// TIA Portal V17 export
// export: Created 2023-09-06T09:59:09.1457623Z, ExportSetting WithDefaults, DisplayName Totally Integrated Automation Portal, DisplayVersion V17 Update 6, DisplayName TIA Portal Openness, DisplayVersion V17 Update 6, DisplayName TIA Portal Teamcenter Gateway, DisplayVersion V17 Update 6, DisplayName TIA Portal Version Control Interface, DisplayVersion V17, DisplayName Simotion SCOUT TIA, DisplayVersion 5.4.3.0, DisplayName TIA Portal Test Suite Advanced, DisplayVersion V17 Update 1, DisplayName SIMOCODE ES, DisplayVersion V17 Update 5, DisplayName SINAMICS Startdrive Advanced, DisplayVersion V17 SP1, DisplayName SINAMICS Startdrive G130, G150, S120, S150, SINAMICS MV, S210, DisplayVersion V17 SP1, DisplayName SINAMICS Startdrive G110M, G120, G120C, G120D, G120P, G115D, DisplayVersion V17 SP1, DisplayName SIRIUS Safety ES, DisplayVersion V17 Update 5, DisplayName STEP 7 Professional, DisplayVersion V17 Update 6, DisplayName STEP 7 CFC, DisplayVersion V17 Update 1, DisplayName STEP 7 Safety, DisplayVersion V17 Update 6, DisplayName WinCC Advanced, DisplayVersion V17 Update 6, DisplayName SIMATIC Visualization Architect, DisplayVersion V17 Update 5
FUNCTION "05_Output Feedback" : Void   // FC6, F_FBD
TITLE = Manage Safety Outputs
{ S7_Optimized_Access := 'TRUE' }
VERSION : 0.1
// stored: AutoNumber true, IsIECCheckEnabled false, UDAEnableTagReadback false
   VAR_TEMP
      DU_EX : Bool;
      ISPC_EX : Bool;
      ZONE_EX : Bool;
   END_VAR
BEGIN

REGION Network 1: Area S1 =SC01+DU001/DU019.EL001 DRIVE UNIT DU001/DU019
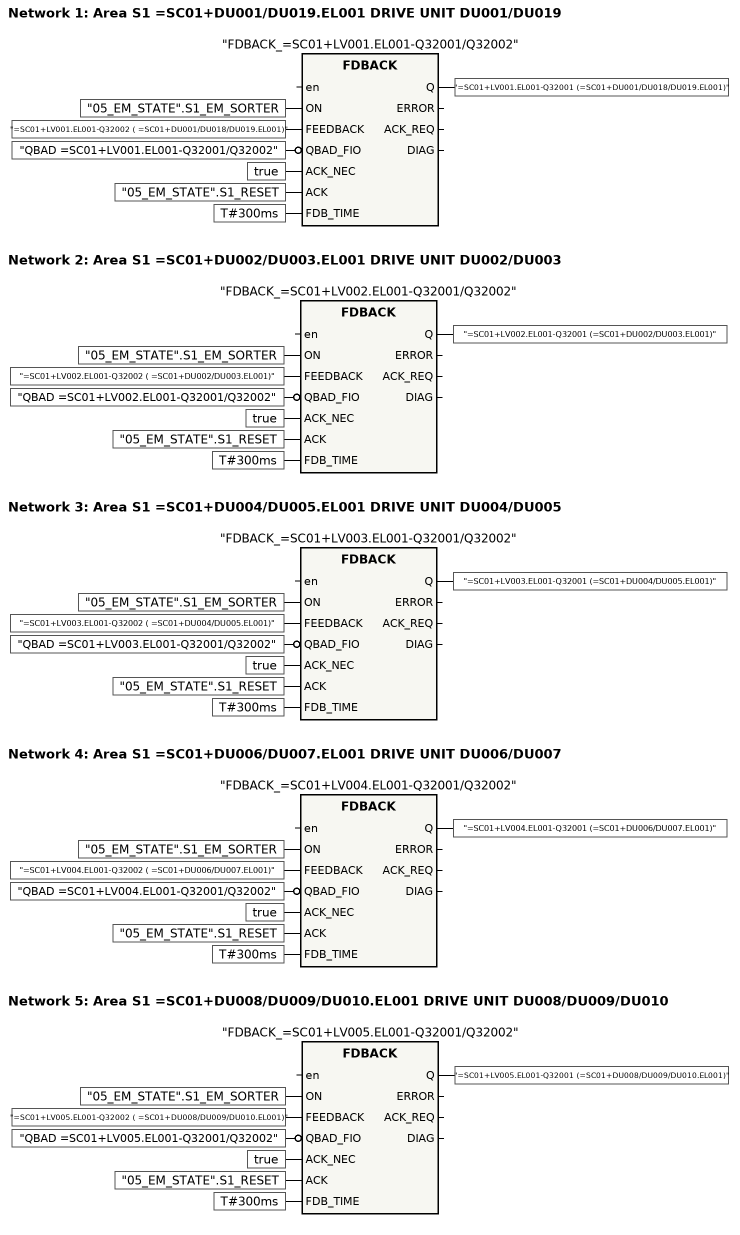
   "FDBACK_=SC01+LV001.EL001-Q32001/Q32002"(ON := "05_EM_STATE".S1_EM_SORTER,   // FDBACK
                           FEEDBACK := "=SC01+LV001.EL001-Q32002 ( =SC01+DU001/DU018/DU019.EL001)",
                           QBAD_FIO := NOT "QBAD =SC01+LV001.EL001-Q32001/Q32002",
                           ACK_NEC := true,
                           ACK := "05_EM_STATE".S1_RESET,
                           FDB_TIME := T#300ms,
                           Q => "=SC01+LV001.EL001-Q32001 (=SC01+DU001/DU018/DU019.EL001)");
END_REGION

REGION Network 2: Area S1 =SC01+DU002/DU003.EL001 DRIVE UNIT DU002/DU003
   "FDBACK_=SC01+LV002.EL001-Q32001/Q32002"(ON := "05_EM_STATE".S1_EM_SORTER,   // FDBACK
                           FEEDBACK := "=SC01+LV002.EL001-Q32002 ( =SC01+DU002/DU003.EL001)",
                           QBAD_FIO := NOT "QBAD =SC01+LV002.EL001-Q32001/Q32002",
                           ACK_NEC := true,
                           ACK := "05_EM_STATE".S1_RESET,
                           FDB_TIME := T#300ms,
                           Q => "=SC01+LV002.EL001-Q32001 (=SC01+DU002/DU003.EL001)");
END_REGION

REGION Network 3: Area S1 =SC01+DU004/DU005.EL001 DRIVE UNIT DU004/DU005
   "FDBACK_=SC01+LV003.EL001-Q32001/Q32002"(ON := "05_EM_STATE".S1_EM_SORTER,   // FDBACK
                           FEEDBACK := "=SC01+LV003.EL001-Q32002 ( =SC01+DU004/DU005.EL001)",
                           QBAD_FIO := NOT "QBAD =SC01+LV003.EL001-Q32001/Q32002",
                           ACK_NEC := true,
                           ACK := "05_EM_STATE".S1_RESET,
                           FDB_TIME := T#300ms,
                           Q => "=SC01+LV003.EL001-Q32001 (=SC01+DU004/DU005.EL001)");
END_REGION

REGION Network 4: Area S1 =SC01+DU006/DU007.EL001 DRIVE UNIT DU006/DU007
   "FDBACK_=SC01+LV004.EL001-Q32001/Q32002"(ON := "05_EM_STATE".S1_EM_SORTER,   // FDBACK
                           FEEDBACK := "=SC01+LV004.EL001-Q32002 ( =SC01+DU006/DU007.EL001)",
                           QBAD_FIO := NOT "QBAD =SC01+LV004.EL001-Q32001/Q32002",
                           ACK_NEC := true,
                           ACK := "05_EM_STATE".S1_RESET,
                           FDB_TIME := T#300ms,
                           Q => "=SC01+LV004.EL001-Q32001 (=SC01+DU006/DU007.EL001)");
END_REGION

REGION Network 5: Area S1 =SC01+DU008/DU009/DU010.EL001 DRIVE UNIT DU008/DU009/DU010
   "FDBACK_=SC01+LV005.EL001-Q32001/Q32002"(ON := "05_EM_STATE".S1_EM_SORTER,   // FDBACK
                           FEEDBACK := "=SC01+LV005.EL001-Q32002 ( =SC01+DU008/DU009/DU010.EL001)",
                           QBAD_FIO := NOT "QBAD =SC01+LV005.EL001-Q32001/Q32002",
                           ACK_NEC := true,
                           ACK := "05_EM_STATE".S1_RESET,
                           FDB_TIME := T#300ms,
                           Q => "=SC01+LV005.EL001-Q32001 (=SC01+DU008/DU009/DU010.EL001)");
END_REGION

REGION Network 6: Area S1 =SC01+DU011/DU012/DU013.EL001 DRIVE UNIT DU011/DU012/DU013
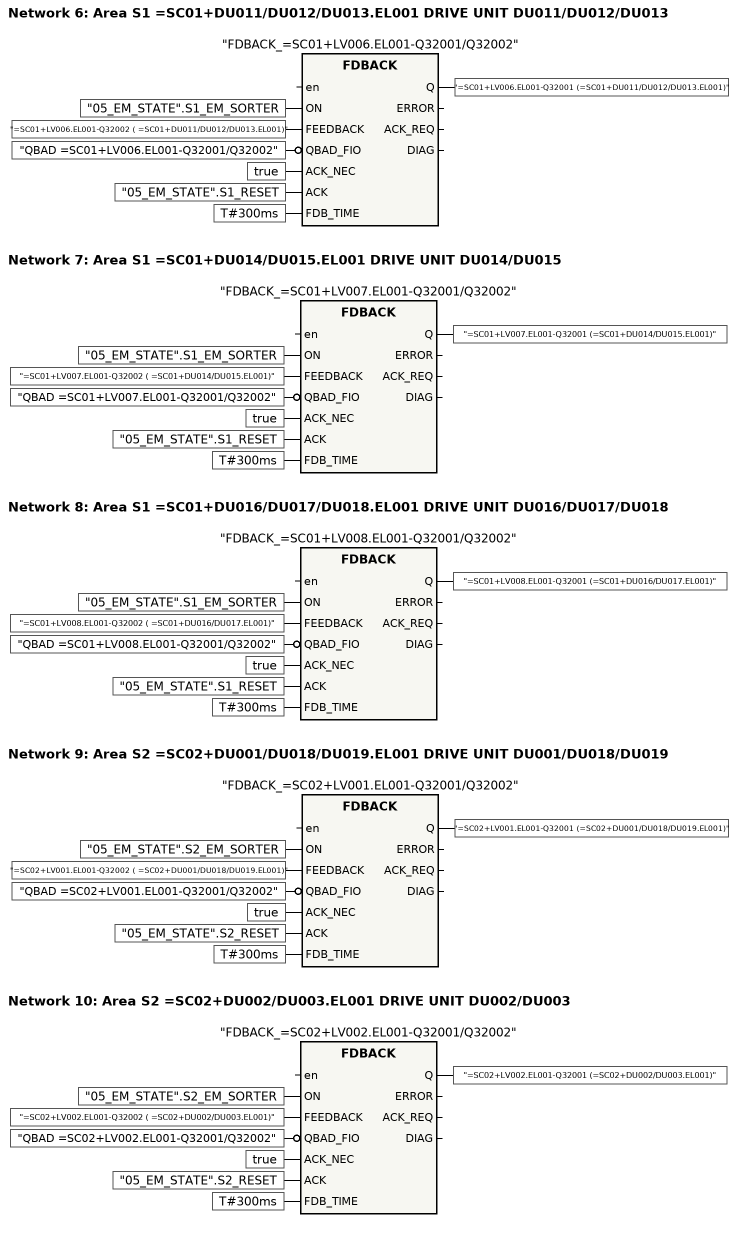
   "FDBACK_=SC01+LV006.EL001-Q32001/Q32002"(ON := "05_EM_STATE".S1_EM_SORTER,   // FDBACK
                           FEEDBACK := "=SC01+LV006.EL001-Q32002 ( =SC01+DU011/DU012/DU013.EL001)",
                           QBAD_FIO := NOT "QBAD =SC01+LV006.EL001-Q32001/Q32002",
                           ACK_NEC := true,
                           ACK := "05_EM_STATE".S1_RESET,
                           FDB_TIME := T#300ms,
                           Q => "=SC01+LV006.EL001-Q32001 (=SC01+DU011/DU012/DU013.EL001)");
END_REGION

REGION Network 7: Area S1 =SC01+DU014/DU015.EL001 DRIVE UNIT DU014/DU015
   "FDBACK_=SC01+LV007.EL001-Q32001/Q32002"(ON := "05_EM_STATE".S1_EM_SORTER,   // FDBACK
                           FEEDBACK := "=SC01+LV007.EL001-Q32002 ( =SC01+DU014/DU015.EL001)",
                           QBAD_FIO := NOT "QBAD =SC01+LV007.EL001-Q32001/Q32002",
                           ACK_NEC := true,
                           ACK := "05_EM_STATE".S1_RESET,
                           FDB_TIME := T#300ms,
                           Q => "=SC01+LV007.EL001-Q32001 (=SC01+DU014/DU015.EL001)");
END_REGION

REGION Network 8: Area S1 =SC01+DU016/DU017/DU018.EL001 DRIVE UNIT DU016/DU017/DU018
   "FDBACK_=SC01+LV008.EL001-Q32001/Q32002"(ON := "05_EM_STATE".S1_EM_SORTER,   // FDBACK
                           FEEDBACK := "=SC01+LV008.EL001-Q32002 ( =SC01+DU016/DU017.EL001)",
                           QBAD_FIO := NOT "QBAD =SC01+LV008.EL001-Q32001/Q32002",
                           ACK_NEC := true,
                           ACK := "05_EM_STATE".S1_RESET,
                           FDB_TIME := T#300ms,
                           Q => "=SC01+LV008.EL001-Q32001 (=SC01+DU016/DU017.EL001)");
END_REGION

REGION Network 9: Area S2 =SC02+DU001/DU018/DU019.EL001 DRIVE UNIT DU001/DU018/DU019
   "FDBACK_=SC02+LV001.EL001-Q32001/Q32002"(ON := "05_EM_STATE".S2_EM_SORTER,   // FDBACK
                           FEEDBACK := "=SC02+LV001.EL001-Q32002 ( =SC02+DU001/DU018/DU019.EL001)",
                           QBAD_FIO := NOT "QBAD =SC02+LV001.EL001-Q32001/Q32002",
                           ACK_NEC := true,
                           ACK := "05_EM_STATE".S2_RESET,
                           FDB_TIME := T#300ms,
                           Q => "=SC02+LV001.EL001-Q32001 (=SC02+DU001/DU018/DU019.EL001)");
END_REGION

REGION Network 10: Area S2 =SC02+DU002/DU003.EL001 DRIVE UNIT DU002/DU003
   "FDBACK_=SC02+LV002.EL001-Q32001/Q32002"(ON := "05_EM_STATE".S2_EM_SORTER,   // FDBACK
                           FEEDBACK := "=SC02+LV002.EL001-Q32002 ( =SC02+DU002/DU003.EL001)",
                           QBAD_FIO := NOT "QBAD =SC02+LV002.EL001-Q32001/Q32002",
                           ACK_NEC := true,
                           ACK := "05_EM_STATE".S2_RESET,
                           FDB_TIME := T#300ms,
                           Q => "=SC02+LV002.EL001-Q32001 (=SC02+DU002/DU003.EL001)");
END_REGION

REGION Network 11: Area S2 =SC02+DU004/DU005.EL001 DRIVE UNIT DU004/DU005
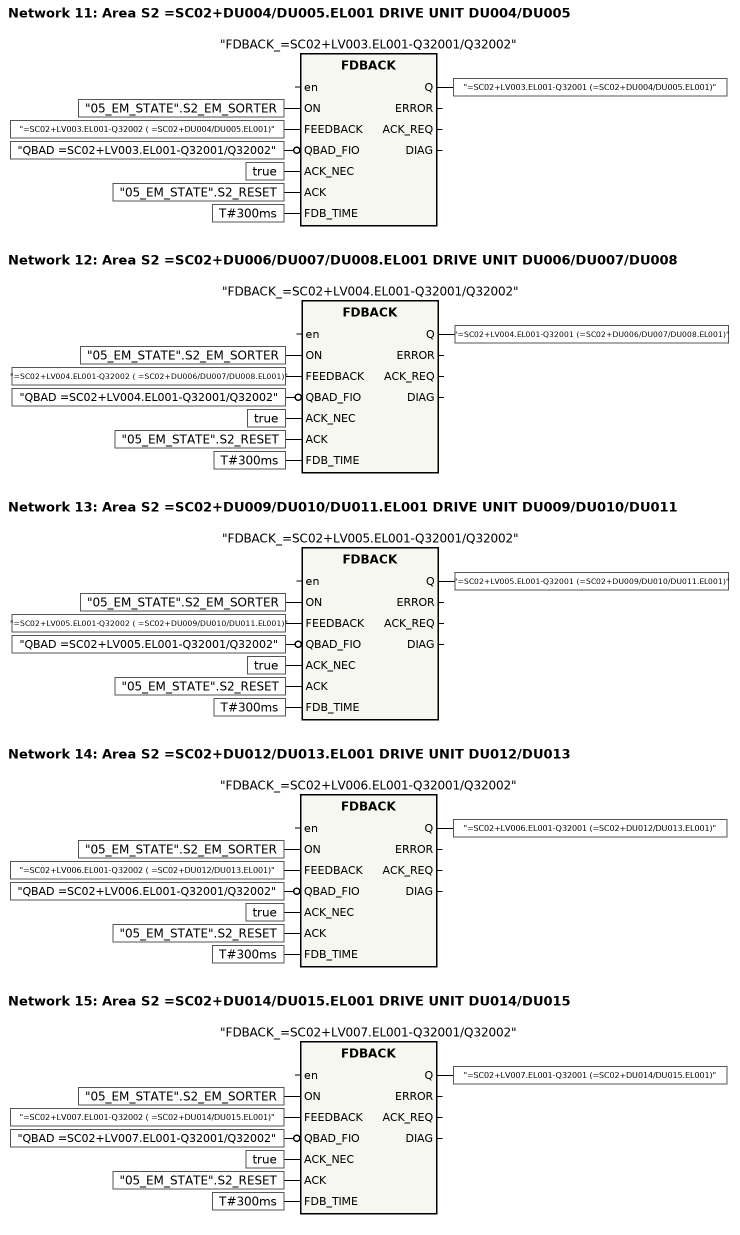
   "FDBACK_=SC02+LV003.EL001-Q32001/Q32002"(ON := "05_EM_STATE".S2_EM_SORTER,   // FDBACK
                           FEEDBACK := "=SC02+LV003.EL001-Q32002 ( =SC02+DU004/DU005.EL001)",
                           QBAD_FIO := NOT "QBAD =SC02+LV003.EL001-Q32001/Q32002",
                           ACK_NEC := true,
                           ACK := "05_EM_STATE".S2_RESET,
                           FDB_TIME := T#300ms,
                           Q => "=SC02+LV003.EL001-Q32001 (=SC02+DU004/DU005.EL001)");
END_REGION

REGION Network 12: Area S2 =SC02+DU006/DU007/DU008.EL001 DRIVE UNIT DU006/DU007/DU008
   "FDBACK_=SC02+LV004.EL001-Q32001/Q32002"(ON := "05_EM_STATE".S2_EM_SORTER,   // FDBACK
                           FEEDBACK := "=SC02+LV004.EL001-Q32002 ( =SC02+DU006/DU007/DU008.EL001)",
                           QBAD_FIO := NOT "QBAD =SC02+LV004.EL001-Q32001/Q32002",
                           ACK_NEC := true,
                           ACK := "05_EM_STATE".S2_RESET,
                           FDB_TIME := T#300ms,
                           Q => "=SC02+LV004.EL001-Q32001 (=SC02+DU006/DU007/DU008.EL001)");
END_REGION

REGION Network 13: Area S2 =SC02+DU009/DU010/DU011.EL001 DRIVE UNIT DU009/DU010/DU011
   "FDBACK_=SC02+LV005.EL001-Q32001/Q32002"(ON := "05_EM_STATE".S2_EM_SORTER,   // FDBACK
                           FEEDBACK := "=SC02+LV005.EL001-Q32002 ( =SC02+DU009/DU010/DU011.EL001)",
                           QBAD_FIO := NOT "QBAD =SC02+LV005.EL001-Q32001/Q32002",
                           ACK_NEC := true,
                           ACK := "05_EM_STATE".S2_RESET,
                           FDB_TIME := T#300ms,
                           Q => "=SC02+LV005.EL001-Q32001 (=SC02+DU009/DU010/DU011.EL001)");
END_REGION

REGION Network 14: Area S2 =SC02+DU012/DU013.EL001 DRIVE UNIT DU012/DU013
   "FDBACK_=SC02+LV006.EL001-Q32001/Q32002"(ON := "05_EM_STATE".S2_EM_SORTER,   // FDBACK
                           FEEDBACK := "=SC02+LV006.EL001-Q32002 ( =SC02+DU012/DU013.EL001)",
                           QBAD_FIO := NOT "QBAD =SC02+LV006.EL001-Q32001/Q32002",
                           ACK_NEC := true,
                           ACK := "05_EM_STATE".S2_RESET,
                           FDB_TIME := T#300ms,
                           Q => "=SC02+LV006.EL001-Q32001 (=SC02+DU012/DU013.EL001)");
END_REGION

REGION Network 15: Area S2 =SC02+DU014/DU015.EL001 DRIVE UNIT DU014/DU015
   "FDBACK_=SC02+LV007.EL001-Q32001/Q32002"(ON := "05_EM_STATE".S2_EM_SORTER,   // FDBACK
                           FEEDBACK := "=SC02+LV007.EL001-Q32002 ( =SC02+DU014/DU015.EL001)",
                           QBAD_FIO := NOT "QBAD =SC02+LV007.EL001-Q32001/Q32002",
                           ACK_NEC := true,
                           ACK := "05_EM_STATE".S2_RESET,
                           FDB_TIME := T#300ms,
                           Q => "=SC02+LV007.EL001-Q32001 (=SC02+DU014/DU015.EL001)");
END_REGION

REGION Network 16: Area S2 =SC02+DU016/DU017.EL001 DRIVE UNIT DU016/DU017
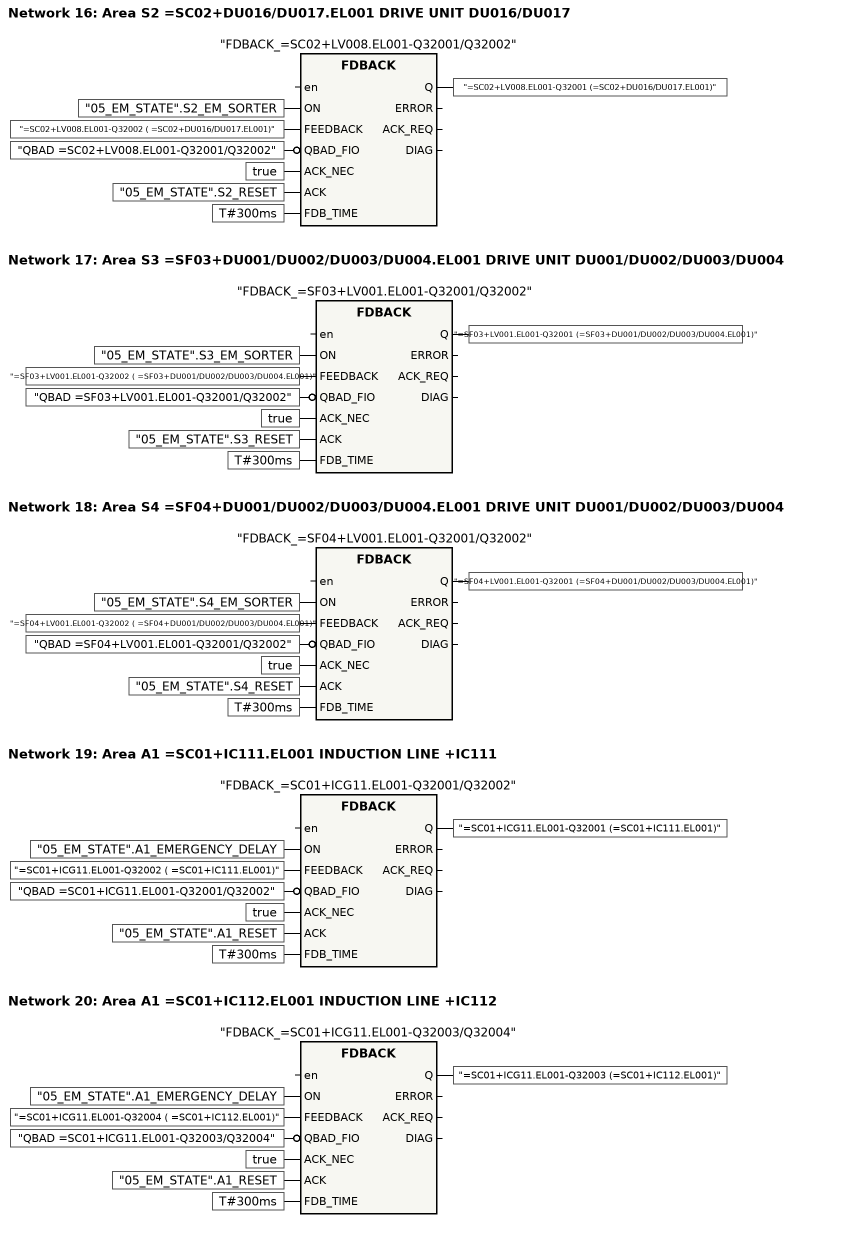
   "FDBACK_=SC02+LV008.EL001-Q32001/Q32002"(ON := "05_EM_STATE".S2_EM_SORTER,   // FDBACK
                           FEEDBACK := "=SC02+LV008.EL001-Q32002 ( =SC02+DU016/DU017.EL001)",
                           QBAD_FIO := NOT "QBAD =SC02+LV008.EL001-Q32001/Q32002",
                           ACK_NEC := true,
                           ACK := "05_EM_STATE".S2_RESET,
                           FDB_TIME := T#300ms,
                           Q => "=SC02+LV008.EL001-Q32001 (=SC02+DU016/DU017.EL001)");
END_REGION

REGION Network 17: Area S3 =SF03+DU001/DU002/DU003/DU004.EL001 DRIVE UNIT DU001/DU002/DU003/DU004
   "FDBACK_=SF03+LV001.EL001-Q32001/Q32002"(ON := "05_EM_STATE".S3_EM_SORTER,   // FDBACK
                           FEEDBACK := "=SF03+LV001.EL001-Q32002 ( =SF03+DU001/DU002/DU003/DU004.EL001)",
                           QBAD_FIO := NOT "QBAD =SF03+LV001.EL001-Q32001/Q32002",
                           ACK_NEC := true,
                           ACK := "05_EM_STATE".S3_RESET,
                           FDB_TIME := T#300ms,
                           Q => "=SF03+LV001.EL001-Q32001 (=SF03+DU001/DU002/DU003/DU004.EL001)");
END_REGION

REGION Network 18: Area S4 =SF04+DU001/DU002/DU003/DU004.EL001 DRIVE UNIT DU001/DU002/DU003/DU004
   "FDBACK_=SF04+LV001.EL001-Q32001/Q32002"(ON := "05_EM_STATE".S4_EM_SORTER,   // FDBACK
                           FEEDBACK := "=SF04+LV001.EL001-Q32002 ( =SF04+DU001/DU002/DU003/DU004.EL001)",
                           QBAD_FIO := NOT "QBAD =SF04+LV001.EL001-Q32001/Q32002",
                           ACK_NEC := true,
                           ACK := "05_EM_STATE".S4_RESET,
                           FDB_TIME := T#300ms,
                           Q => "=SF04+LV001.EL001-Q32001 (=SF04+DU001/DU002/DU003/DU004.EL001)");
END_REGION

REGION Network 19: Area A1 =SC01+IC111.EL001 INDUCTION LINE +IC111
   "FDBACK_=SC01+ICG11.EL001-Q32001/Q32002"(ON := "05_EM_STATE".A1_EMERGENCY_DELAY,   // FDBACK
                           FEEDBACK := "=SC01+ICG11.EL001-Q32002 ( =SC01+IC111.EL001)",
                           QBAD_FIO := NOT "QBAD =SC01+ICG11.EL001-Q32001/Q32002",
                           ACK_NEC := true,
                           ACK := "05_EM_STATE".A1_RESET,
                           FDB_TIME := T#300ms,
                           Q => "=SC01+ICG11.EL001-Q32001 (=SC01+IC111.EL001)");
END_REGION

REGION Network 20: Area A1 =SC01+IC112.EL001 INDUCTION LINE +IC112
   "FDBACK_=SC01+ICG11.EL001-Q32003/Q32004"(ON := "05_EM_STATE".A1_EMERGENCY_DELAY,   // FDBACK
                           FEEDBACK := "=SC01+ICG11.EL001-Q32004 ( =SC01+IC112.EL001)",
                           QBAD_FIO := NOT "QBAD =SC01+ICG11.EL001-Q32003/Q32004",
                           ACK_NEC := true,
                           ACK := "05_EM_STATE".A1_RESET,
                           FDB_TIME := T#300ms,
                           Q => "=SC01+ICG11.EL001-Q32003 (=SC01+IC112.EL001)");
END_REGION

REGION Network 21: Area A1 =SC01+IC113.EL001 INDUCTION LINE +IC113
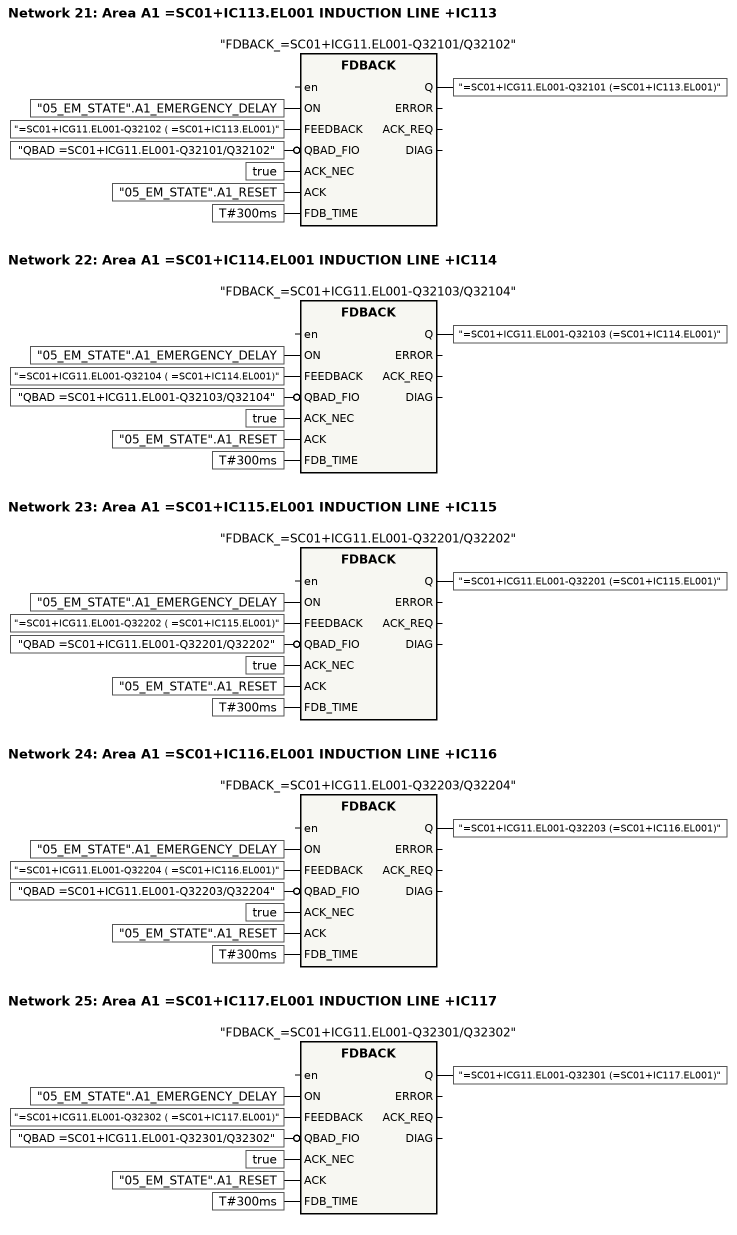
   "FDBACK_=SC01+ICG11.EL001-Q32101/Q32102"(ON := "05_EM_STATE".A1_EMERGENCY_DELAY,   // FDBACK
                           FEEDBACK := "=SC01+ICG11.EL001-Q32102 ( =SC01+IC113.EL001)",
                           QBAD_FIO := NOT "QBAD =SC01+ICG11.EL001-Q32101/Q32102",
                           ACK_NEC := true,
                           ACK := "05_EM_STATE".A1_RESET,
                           FDB_TIME := T#300ms,
                           Q => "=SC01+ICG11.EL001-Q32101 (=SC01+IC113.EL001)");
END_REGION

REGION Network 22: Area A1 =SC01+IC114.EL001 INDUCTION LINE +IC114
   "FDBACK_=SC01+ICG11.EL001-Q32103/Q32104"(ON := "05_EM_STATE".A1_EMERGENCY_DELAY,   // FDBACK
                           FEEDBACK := "=SC01+ICG11.EL001-Q32104 ( =SC01+IC114.EL001)",
                           QBAD_FIO := NOT "QBAD =SC01+ICG11.EL001-Q32103/Q32104",
                           ACK_NEC := true,
                           ACK := "05_EM_STATE".A1_RESET,
                           FDB_TIME := T#300ms,
                           Q => "=SC01+ICG11.EL001-Q32103 (=SC01+IC114.EL001)");
END_REGION

REGION Network 23: Area A1 =SC01+IC115.EL001 INDUCTION LINE +IC115
   "FDBACK_=SC01+ICG11.EL001-Q32201/Q32202"(ON := "05_EM_STATE".A1_EMERGENCY_DELAY,   // FDBACK
                           FEEDBACK := "=SC01+ICG11.EL001-Q32202 ( =SC01+IC115.EL001)",
                           QBAD_FIO := NOT "QBAD =SC01+ICG11.EL001-Q32201/Q32202",
                           ACK_NEC := true,
                           ACK := "05_EM_STATE".A1_RESET,
                           FDB_TIME := T#300ms,
                           Q => "=SC01+ICG11.EL001-Q32201 (=SC01+IC115.EL001)");
END_REGION

REGION Network 24: Area A1 =SC01+IC116.EL001 INDUCTION LINE +IC116
   "FDBACK_=SC01+ICG11.EL001-Q32203/Q32204"(ON := "05_EM_STATE".A1_EMERGENCY_DELAY,   // FDBACK
                           FEEDBACK := "=SC01+ICG11.EL001-Q32204 ( =SC01+IC116.EL001)",
                           QBAD_FIO := NOT "QBAD =SC01+ICG11.EL001-Q32203/Q32204",
                           ACK_NEC := true,
                           ACK := "05_EM_STATE".A1_RESET,
                           FDB_TIME := T#300ms,
                           Q => "=SC01+ICG11.EL001-Q32203 (=SC01+IC116.EL001)");
END_REGION

REGION Network 25: Area A1 =SC01+IC117.EL001 INDUCTION LINE +IC117
   "FDBACK_=SC01+ICG11.EL001-Q32301/Q32302"(ON := "05_EM_STATE".A1_EMERGENCY_DELAY,   // FDBACK
                           FEEDBACK := "=SC01+ICG11.EL001-Q32302 ( =SC01+IC117.EL001)",
                           QBAD_FIO := NOT "QBAD =SC01+ICG11.EL001-Q32301/Q32302",
                           ACK_NEC := true,
                           ACK := "05_EM_STATE".A1_RESET,
                           FDB_TIME := T#300ms,
                           Q => "=SC01+ICG11.EL001-Q32301 (=SC01+IC117.EL001)");
END_REGION

REGION Network 26: Area A1 =SC01+IC121.EL001 INDUCTION LINE +IC121
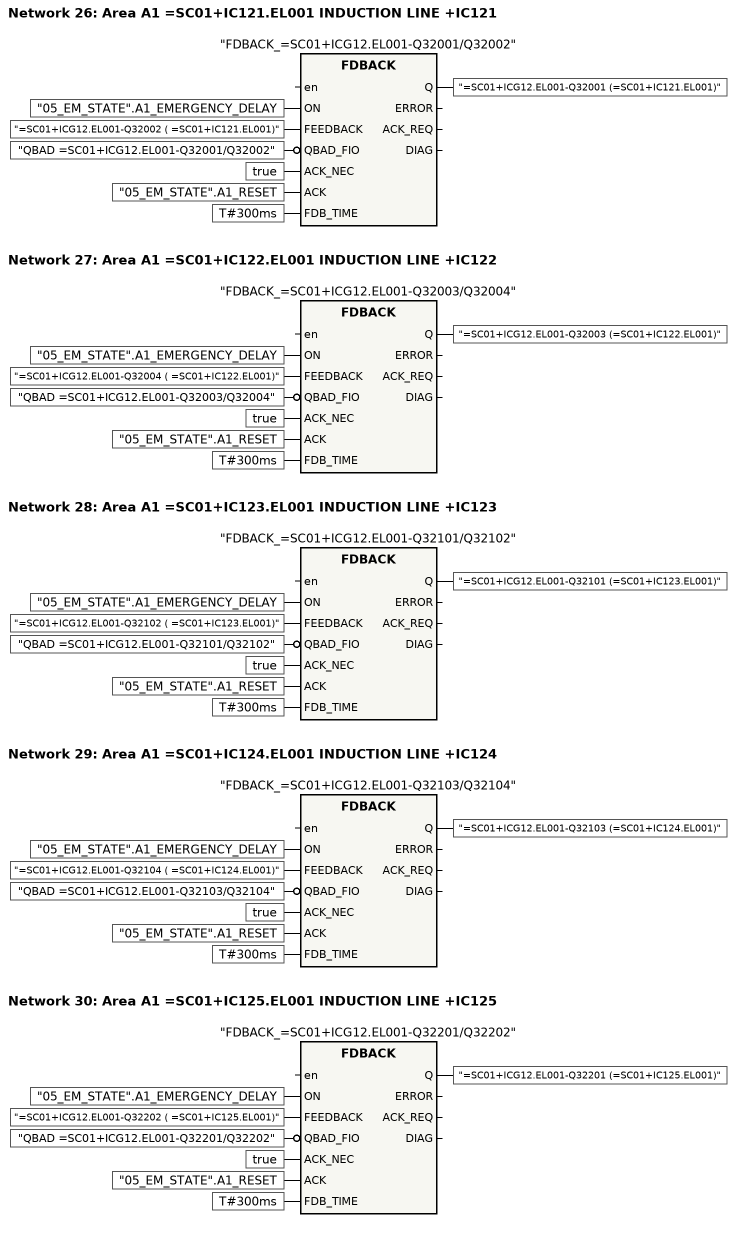
   "FDBACK_=SC01+ICG12.EL001-Q32001/Q32002"(ON := "05_EM_STATE".A1_EMERGENCY_DELAY,   // FDBACK
                           FEEDBACK := "=SC01+ICG12.EL001-Q32002 ( =SC01+IC121.EL001)",
                           QBAD_FIO := NOT "QBAD =SC01+ICG12.EL001-Q32001/Q32002",
                           ACK_NEC := true,
                           ACK := "05_EM_STATE".A1_RESET,
                           FDB_TIME := T#300ms,
                           Q => "=SC01+ICG12.EL001-Q32001 (=SC01+IC121.EL001)");
END_REGION

REGION Network 27: Area A1 =SC01+IC122.EL001 INDUCTION LINE +IC122
   "FDBACK_=SC01+ICG12.EL001-Q32003/Q32004"(ON := "05_EM_STATE".A1_EMERGENCY_DELAY,   // FDBACK
                           FEEDBACK := "=SC01+ICG12.EL001-Q32004 ( =SC01+IC122.EL001)",
                           QBAD_FIO := NOT "QBAD =SC01+ICG12.EL001-Q32003/Q32004",
                           ACK_NEC := true,
                           ACK := "05_EM_STATE".A1_RESET,
                           FDB_TIME := T#300ms,
                           Q => "=SC01+ICG12.EL001-Q32003 (=SC01+IC122.EL001)");
END_REGION

REGION Network 28: Area A1 =SC01+IC123.EL001 INDUCTION LINE +IC123
   "FDBACK_=SC01+ICG12.EL001-Q32101/Q32102"(ON := "05_EM_STATE".A1_EMERGENCY_DELAY,   // FDBACK
                           FEEDBACK := "=SC01+ICG12.EL001-Q32102 ( =SC01+IC123.EL001)",
                           QBAD_FIO := NOT "QBAD =SC01+ICG12.EL001-Q32101/Q32102",
                           ACK_NEC := true,
                           ACK := "05_EM_STATE".A1_RESET,
                           FDB_TIME := T#300ms,
                           Q => "=SC01+ICG12.EL001-Q32101 (=SC01+IC123.EL001)");
END_REGION

REGION Network 29: Area A1 =SC01+IC124.EL001 INDUCTION LINE +IC124
   "FDBACK_=SC01+ICG12.EL001-Q32103/Q32104"(ON := "05_EM_STATE".A1_EMERGENCY_DELAY,   // FDBACK
                           FEEDBACK := "=SC01+ICG12.EL001-Q32104 ( =SC01+IC124.EL001)",
                           QBAD_FIO := NOT "QBAD =SC01+ICG12.EL001-Q32103/Q32104",
                           ACK_NEC := true,
                           ACK := "05_EM_STATE".A1_RESET,
                           FDB_TIME := T#300ms,
                           Q => "=SC01+ICG12.EL001-Q32103 (=SC01+IC124.EL001)");
END_REGION

REGION Network 30: Area A1 =SC01+IC125.EL001 INDUCTION LINE +IC125
   "FDBACK_=SC01+ICG12.EL001-Q32201/Q32202"(ON := "05_EM_STATE".A1_EMERGENCY_DELAY,   // FDBACK
                           FEEDBACK := "=SC01+ICG12.EL001-Q32202 ( =SC01+IC125.EL001)",
                           QBAD_FIO := NOT "QBAD =SC01+ICG12.EL001-Q32201/Q32202",
                           ACK_NEC := true,
                           ACK := "05_EM_STATE".A1_RESET,
                           FDB_TIME := T#300ms,
                           Q => "=SC01+ICG12.EL001-Q32201 (=SC01+IC125.EL001)");
END_REGION

REGION Network 31: Area A1 =SC01+IC126.EL001 INDUCTION LINE +IC126
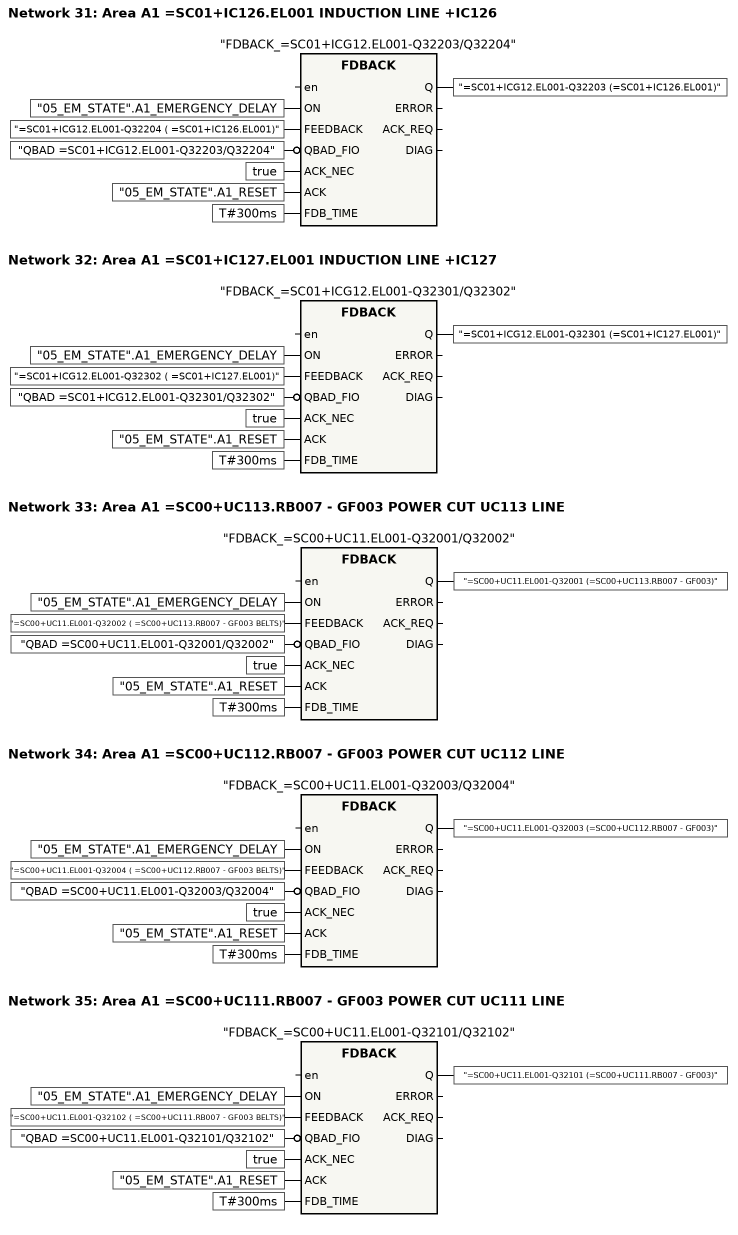
   "FDBACK_=SC01+ICG12.EL001-Q32203/Q32204"(ON := "05_EM_STATE".A1_EMERGENCY_DELAY,   // FDBACK
                           FEEDBACK := "=SC01+ICG12.EL001-Q32204 ( =SC01+IC126.EL001)",
                           QBAD_FIO := NOT "QBAD =SC01+ICG12.EL001-Q32203/Q32204",
                           ACK_NEC := true,
                           ACK := "05_EM_STATE".A1_RESET,
                           FDB_TIME := T#300ms,
                           Q => "=SC01+ICG12.EL001-Q32203 (=SC01+IC126.EL001)");
END_REGION

REGION Network 32: Area A1 =SC01+IC127.EL001 INDUCTION LINE +IC127
   "FDBACK_=SC01+ICG12.EL001-Q32301/Q32302"(ON := "05_EM_STATE".A1_EMERGENCY_DELAY,   // FDBACK
                           FEEDBACK := "=SC01+ICG12.EL001-Q32302 ( =SC01+IC127.EL001)",
                           QBAD_FIO := NOT "QBAD =SC01+ICG12.EL001-Q32301/Q32302",
                           ACK_NEC := true,
                           ACK := "05_EM_STATE".A1_RESET,
                           FDB_TIME := T#300ms,
                           Q => "=SC01+ICG12.EL001-Q32301 (=SC01+IC127.EL001)");
END_REGION

REGION Network 33: Area A1 =SC00+UC113.RB007 - GF003 POWER CUT UC113 LINE
   "FDBACK_=SC00+UC11.EL001-Q32001/Q32002"(ON := "05_EM_STATE".A1_EMERGENCY_DELAY,   // FDBACK
                           FEEDBACK := "=SC00+UC11.EL001-Q32002 ( =SC00+UC113.RB007 - GF003 BELTS)",
                           QBAD_FIO := NOT "QBAD =SC00+UC11.EL001-Q32001/Q32002",
                           ACK_NEC := true,
                           ACK := "05_EM_STATE".A1_RESET,
                           FDB_TIME := T#300ms,
                           Q => "=SC00+UC11.EL001-Q32001 (=SC00+UC113.RB007 - GF003)");
END_REGION

REGION Network 34: Area A1 =SC00+UC112.RB007 - GF003 POWER CUT UC112 LINE
   "FDBACK_=SC00+UC11.EL001-Q32003/Q32004"(ON := "05_EM_STATE".A1_EMERGENCY_DELAY,   // FDBACK
                           FEEDBACK := "=SC00+UC11.EL001-Q32004 ( =SC00+UC112.RB007 - GF003 BELTS)",
                           QBAD_FIO := NOT "QBAD =SC00+UC11.EL001-Q32003/Q32004",
                           ACK_NEC := true,
                           ACK := "05_EM_STATE".A1_RESET,
                           FDB_TIME := T#300ms,
                           Q => "=SC00+UC11.EL001-Q32003 (=SC00+UC112.RB007 - GF003)");
END_REGION

REGION Network 35: Area A1 =SC00+UC111.RB007 - GF003 POWER CUT UC111 LINE
   "FDBACK_=SC00+UC11.EL001-Q32101/Q32102"(ON := "05_EM_STATE".A1_EMERGENCY_DELAY,   // FDBACK
                           FEEDBACK := "=SC00+UC11.EL001-Q32102 ( =SC00+UC111.RB007 - GF003 BELTS)",
                           QBAD_FIO := NOT "QBAD =SC00+UC11.EL001-Q32101/Q32102",
                           ACK_NEC := true,
                           ACK := "05_EM_STATE".A1_RESET,
                           FDB_TIME := T#300ms,
                           Q => "=SC00+UC11.EL001-Q32101 (=SC00+UC111.RB007 - GF003)");
END_REGION

REGION Network 36: Area A1 =SC00+UC114.GF007 - GF001 POWER CUT UC114 LINE
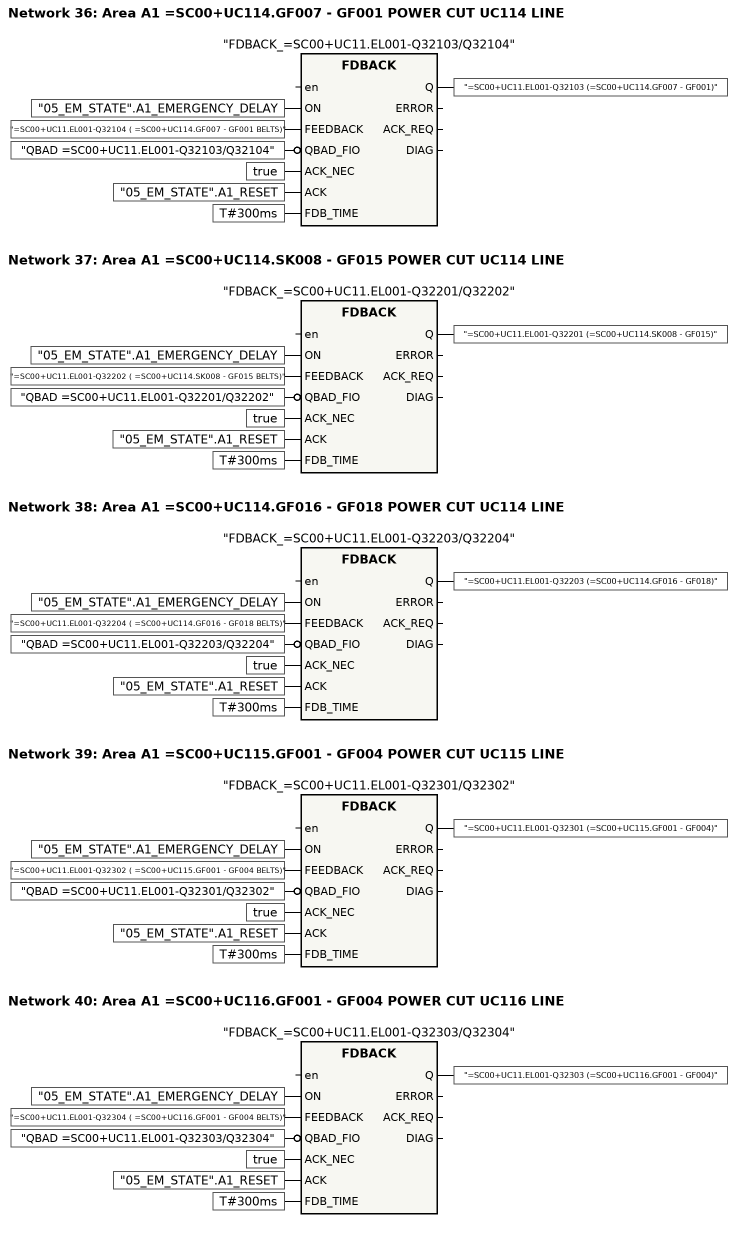
   "FDBACK_=SC00+UC11.EL001-Q32103/Q32104"(ON := "05_EM_STATE".A1_EMERGENCY_DELAY,   // FDBACK
                           FEEDBACK := "=SC00+UC11.EL001-Q32104 ( =SC00+UC114.GF007 - GF001 BELTS)",
                           QBAD_FIO := NOT "QBAD =SC00+UC11.EL001-Q32103/Q32104",
                           ACK_NEC := true,
                           ACK := "05_EM_STATE".A1_RESET,
                           FDB_TIME := T#300ms,
                           Q => "=SC00+UC11.EL001-Q32103 (=SC00+UC114.GF007 - GF001)");
END_REGION

REGION Network 37: Area A1 =SC00+UC114.SK008 - GF015 POWER CUT UC114 LINE
   "FDBACK_=SC00+UC11.EL001-Q32201/Q32202"(ON := "05_EM_STATE".A1_EMERGENCY_DELAY,   // FDBACK
                           FEEDBACK := "=SC00+UC11.EL001-Q32202 ( =SC00+UC114.SK008 - GF015 BELTS)",
                           QBAD_FIO := NOT "QBAD =SC00+UC11.EL001-Q32201/Q32202",
                           ACK_NEC := true,
                           ACK := "05_EM_STATE".A1_RESET,
                           FDB_TIME := T#300ms,
                           Q => "=SC00+UC11.EL001-Q32201 (=SC00+UC114.SK008 - GF015)");
END_REGION

REGION Network 38: Area A1 =SC00+UC114.GF016 - GF018 POWER CUT UC114 LINE
   "FDBACK_=SC00+UC11.EL001-Q32203/Q32204"(ON := "05_EM_STATE".A1_EMERGENCY_DELAY,   // FDBACK
                           FEEDBACK := "=SC00+UC11.EL001-Q32204 ( =SC00+UC114.GF016 - GF018 BELTS)",
                           QBAD_FIO := NOT "QBAD =SC00+UC11.EL001-Q32203/Q32204",
                           ACK_NEC := true,
                           ACK := "05_EM_STATE".A1_RESET,
                           FDB_TIME := T#300ms,
                           Q => "=SC00+UC11.EL001-Q32203 (=SC00+UC114.GF016 - GF018)");
END_REGION

REGION Network 39: Area A1 =SC00+UC115.GF001 - GF004 POWER CUT UC115 LINE
   "FDBACK_=SC00+UC11.EL001-Q32301/Q32302"(ON := "05_EM_STATE".A1_EMERGENCY_DELAY,   // FDBACK
                           FEEDBACK := "=SC00+UC11.EL001-Q32302 ( =SC00+UC115.GF001 - GF004 BELTS)",
                           QBAD_FIO := NOT "QBAD =SC00+UC11.EL001-Q32301/Q32302",
                           ACK_NEC := true,
                           ACK := "05_EM_STATE".A1_RESET,
                           FDB_TIME := T#300ms,
                           Q => "=SC00+UC11.EL001-Q32301 (=SC00+UC115.GF001 - GF004)");
END_REGION

REGION Network 40: Area A1 =SC00+UC116.GF001 - GF004 POWER CUT UC116 LINE
   "FDBACK_=SC00+UC11.EL001-Q32303/Q32304"(ON := "05_EM_STATE".A1_EMERGENCY_DELAY,   // FDBACK
                           FEEDBACK := "=SC00+UC11.EL001-Q32304 ( =SC00+UC116.GF001 - GF004 BELTS)",
                           QBAD_FIO := NOT "QBAD =SC00+UC11.EL001-Q32303/Q32304",
                           ACK_NEC := true,
                           ACK := "05_EM_STATE".A1_RESET,
                           FDB_TIME := T#300ms,
                           Q => "=SC00+UC11.EL001-Q32303 (=SC00+UC116.GF001 - GF004)");
END_REGION

REGION Network 41: Area A1 =SC00+UC117.RB001 - GF003 POWER CUT UC117 LINE
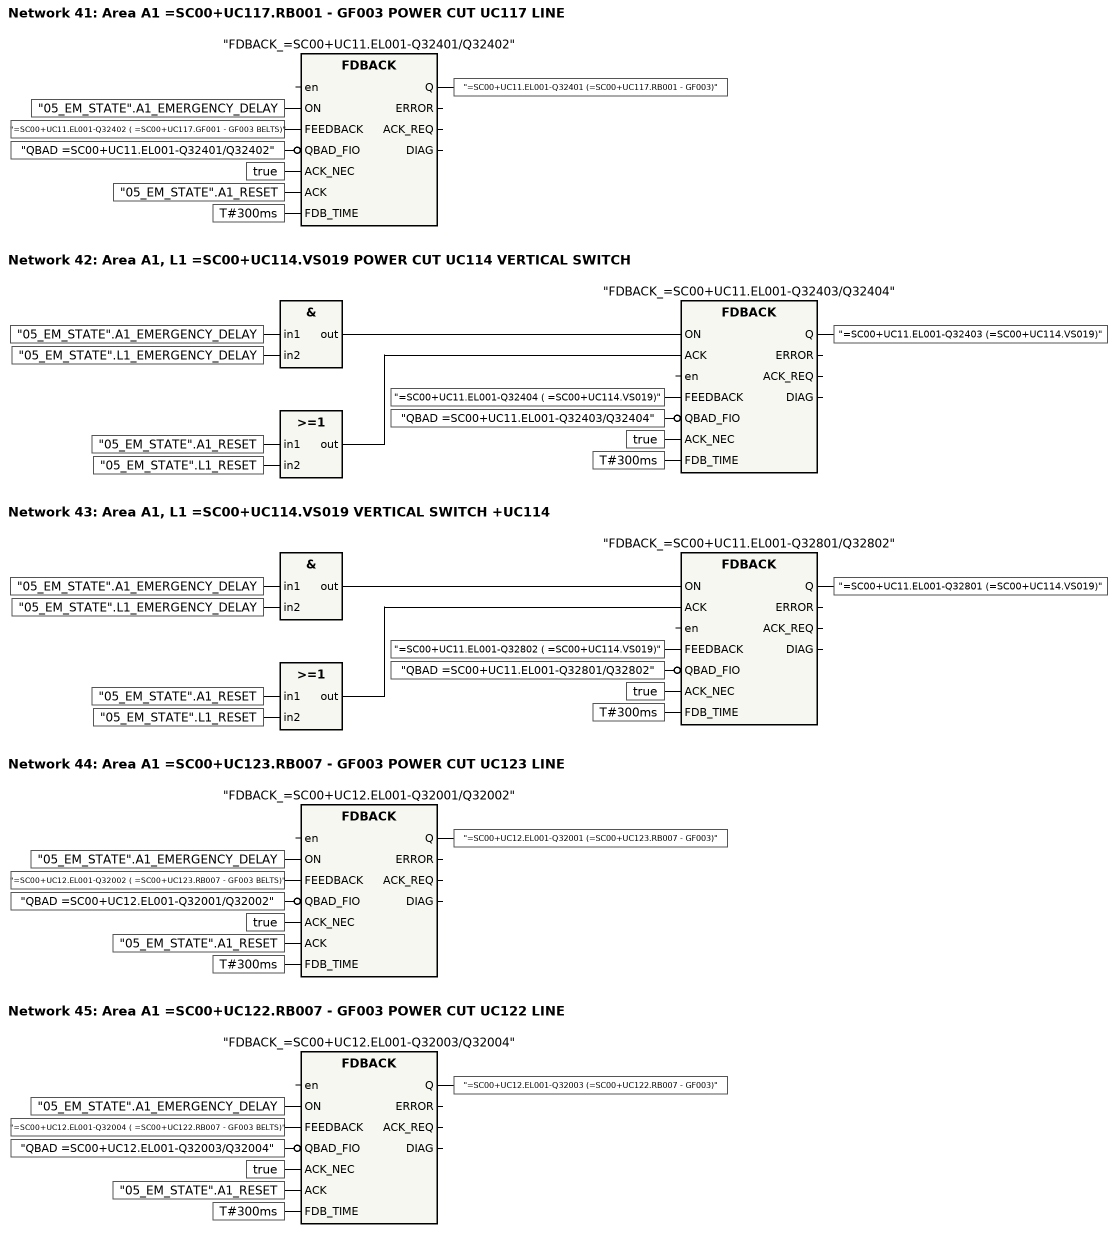
   "FDBACK_=SC00+UC11.EL001-Q32401/Q32402"(ON := "05_EM_STATE".A1_EMERGENCY_DELAY,   // FDBACK
                           FEEDBACK := "=SC00+UC11.EL001-Q32402 ( =SC00+UC117.GF001 - GF003 BELTS)",
                           QBAD_FIO := NOT "QBAD =SC00+UC11.EL001-Q32401/Q32402",
                           ACK_NEC := true,
                           ACK := "05_EM_STATE".A1_RESET,
                           FDB_TIME := T#300ms,
                           Q => "=SC00+UC11.EL001-Q32401 (=SC00+UC117.RB001 - GF003)");
END_REGION

REGION Network 42: Area A1, L1 =SC00+UC114.VS019 POWER CUT UC114 VERTICAL SWITCH
   "FDBACK_=SC00+UC11.EL001-Q32403/Q32404"(ON := "05_EM_STATE".A1_EMERGENCY_DELAY AND "05_EM_STATE".L1_EMERGENCY_DELAY,   // FDBACK
                           ACK := "05_EM_STATE".A1_RESET OR "05_EM_STATE".L1_RESET,
                           FEEDBACK := "=SC00+UC11.EL001-Q32404 ( =SC00+UC114.VS019)",
                           QBAD_FIO := NOT "QBAD =SC00+UC11.EL001-Q32403/Q32404",
                           ACK_NEC := true,
                           FDB_TIME := T#300ms,
                           Q => "=SC00+UC11.EL001-Q32403 (=SC00+UC114.VS019)");
END_REGION

REGION Network 43: Area A1, L1 =SC00+UC114.VS019 VERTICAL SWITCH +UC114
   "FDBACK_=SC00+UC11.EL001-Q32801/Q32802"(ON := "05_EM_STATE".A1_EMERGENCY_DELAY AND "05_EM_STATE".L1_EMERGENCY_DELAY,   // FDBACK
                           ACK := "05_EM_STATE".A1_RESET OR "05_EM_STATE".L1_RESET,
                           FEEDBACK := "=SC00+UC11.EL001-Q32802 ( =SC00+UC114.VS019)",
                           QBAD_FIO := NOT "QBAD =SC00+UC11.EL001-Q32801/Q32802",
                           ACK_NEC := true,
                           FDB_TIME := T#300ms,
                           Q => "=SC00+UC11.EL001-Q32801 (=SC00+UC114.VS019)");
END_REGION

REGION Network 44: Area A1 =SC00+UC123.RB007 - GF003 POWER CUT UC123 LINE
   "FDBACK_=SC00+UC12.EL001-Q32001/Q32002"(ON := "05_EM_STATE".A1_EMERGENCY_DELAY,   // FDBACK
                           FEEDBACK := "=SC00+UC12.EL001-Q32002 ( =SC00+UC123.RB007 - GF003 BELTS)",
                           QBAD_FIO := NOT "QBAD =SC00+UC12.EL001-Q32001/Q32002",
                           ACK_NEC := true,
                           ACK := "05_EM_STATE".A1_RESET,
                           FDB_TIME := T#300ms,
                           Q => "=SC00+UC12.EL001-Q32001 (=SC00+UC123.RB007 - GF003)");
END_REGION

REGION Network 45: Area A1 =SC00+UC122.RB007 - GF003 POWER CUT UC122 LINE
   "FDBACK_=SC00+UC12.EL001-Q32003/Q32004"(ON := "05_EM_STATE".A1_EMERGENCY_DELAY,   // FDBACK
                           FEEDBACK := "=SC00+UC12.EL001-Q32004 ( =SC00+UC122.RB007 - GF003 BELTS)",
                           QBAD_FIO := NOT "QBAD =SC00+UC12.EL001-Q32003/Q32004",
                           ACK_NEC := true,
                           ACK := "05_EM_STATE".A1_RESET,
                           FDB_TIME := T#300ms,
                           Q => "=SC00+UC12.EL001-Q32003 (=SC00+UC122.RB007 - GF003)");
END_REGION

REGION Network 46: Area A1 =SC00+UC121.RB007 - GF003 POWER CUT UC121 LINE
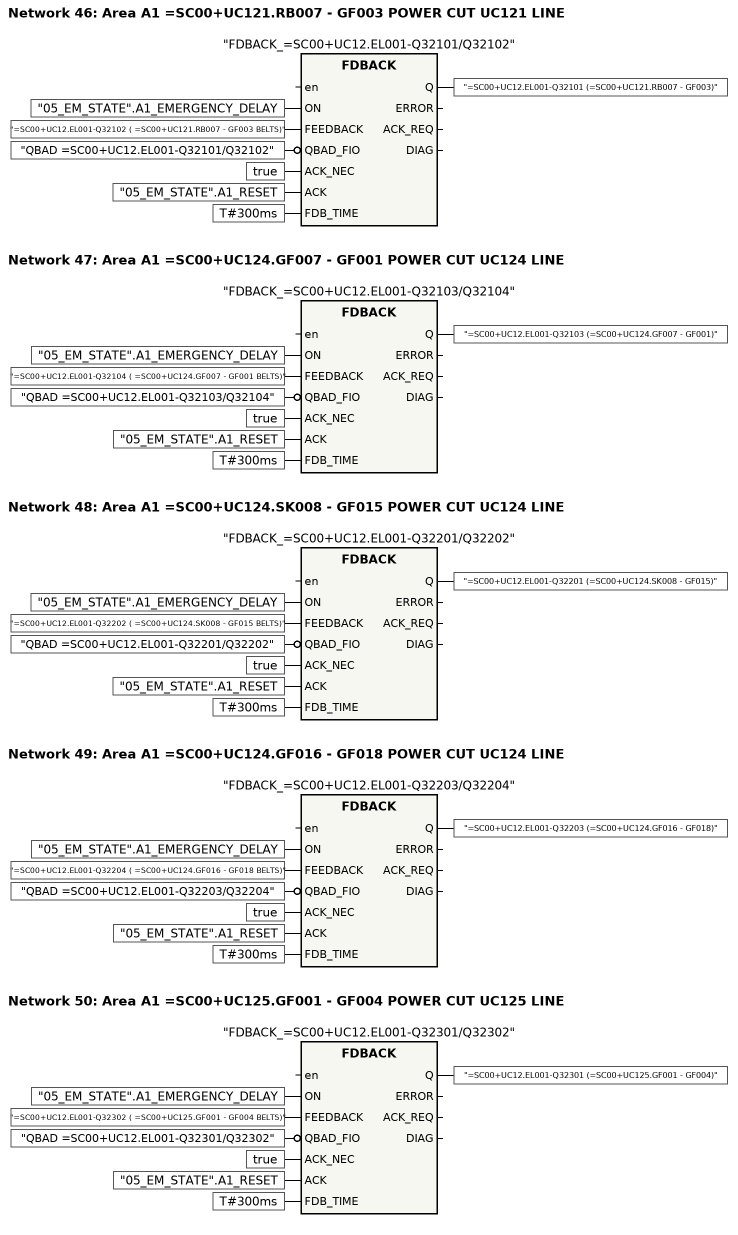
   "FDBACK_=SC00+UC12.EL001-Q32101/Q32102"(ON := "05_EM_STATE".A1_EMERGENCY_DELAY,   // FDBACK
                           FEEDBACK := "=SC00+UC12.EL001-Q32102 ( =SC00+UC121.RB007 - GF003 BELTS)",
                           QBAD_FIO := NOT "QBAD =SC00+UC12.EL001-Q32101/Q32102",
                           ACK_NEC := true,
                           ACK := "05_EM_STATE".A1_RESET,
                           FDB_TIME := T#300ms,
                           Q => "=SC00+UC12.EL001-Q32101 (=SC00+UC121.RB007 - GF003)");
END_REGION

REGION Network 47: Area A1 =SC00+UC124.GF007 - GF001 POWER CUT UC124 LINE
   "FDBACK_=SC00+UC12.EL001-Q32103/Q32104"(ON := "05_EM_STATE".A1_EMERGENCY_DELAY,   // FDBACK
                           FEEDBACK := "=SC00+UC12.EL001-Q32104 ( =SC00+UC124.GF007 - GF001 BELTS)",
                           QBAD_FIO := NOT "QBAD =SC00+UC12.EL001-Q32103/Q32104",
                           ACK_NEC := true,
                           ACK := "05_EM_STATE".A1_RESET,
                           FDB_TIME := T#300ms,
                           Q => "=SC00+UC12.EL001-Q32103 (=SC00+UC124.GF007 - GF001)");
END_REGION

REGION Network 48: Area A1 =SC00+UC124.SK008 - GF015 POWER CUT UC124 LINE
   "FDBACK_=SC00+UC12.EL001-Q32201/Q32202"(ON := "05_EM_STATE".A1_EMERGENCY_DELAY,   // FDBACK
                           FEEDBACK := "=SC00+UC12.EL001-Q32202 ( =SC00+UC124.SK008 - GF015 BELTS)",
                           QBAD_FIO := NOT "QBAD =SC00+UC12.EL001-Q32201/Q32202",
                           ACK_NEC := true,
                           ACK := "05_EM_STATE".A1_RESET,
                           FDB_TIME := T#300ms,
                           Q => "=SC00+UC12.EL001-Q32201 (=SC00+UC124.SK008 - GF015)");
END_REGION

REGION Network 49: Area A1 =SC00+UC124.GF016 - GF018 POWER CUT UC124 LINE
   "FDBACK_=SC00+UC12.EL001-Q32203/Q32204"(ON := "05_EM_STATE".A1_EMERGENCY_DELAY,   // FDBACK
                           FEEDBACK := "=SC00+UC12.EL001-Q32204 ( =SC00+UC124.GF016 - GF018 BELTS)",
                           QBAD_FIO := NOT "QBAD =SC00+UC12.EL001-Q32203/Q32204",
                           ACK_NEC := true,
                           ACK := "05_EM_STATE".A1_RESET,
                           FDB_TIME := T#300ms,
                           Q => "=SC00+UC12.EL001-Q32203 (=SC00+UC124.GF016 - GF018)");
END_REGION

REGION Network 50: Area A1 =SC00+UC125.GF001 - GF004 POWER CUT UC125 LINE
   "FDBACK_=SC00+UC12.EL001-Q32301/Q32302"(ON := "05_EM_STATE".A1_EMERGENCY_DELAY,   // FDBACK
                           FEEDBACK := "=SC00+UC12.EL001-Q32302 ( =SC00+UC125.GF001 - GF004 BELTS)",
                           QBAD_FIO := NOT "QBAD =SC00+UC12.EL001-Q32301/Q32302",
                           ACK_NEC := true,
                           ACK := "05_EM_STATE".A1_RESET,
                           FDB_TIME := T#300ms,
                           Q => "=SC00+UC12.EL001-Q32301 (=SC00+UC125.GF001 - GF004)");
END_REGION

REGION Network 51: Area A1 =SC00+UC126.GF001 - GF004 POWER CUT UC126 LINE
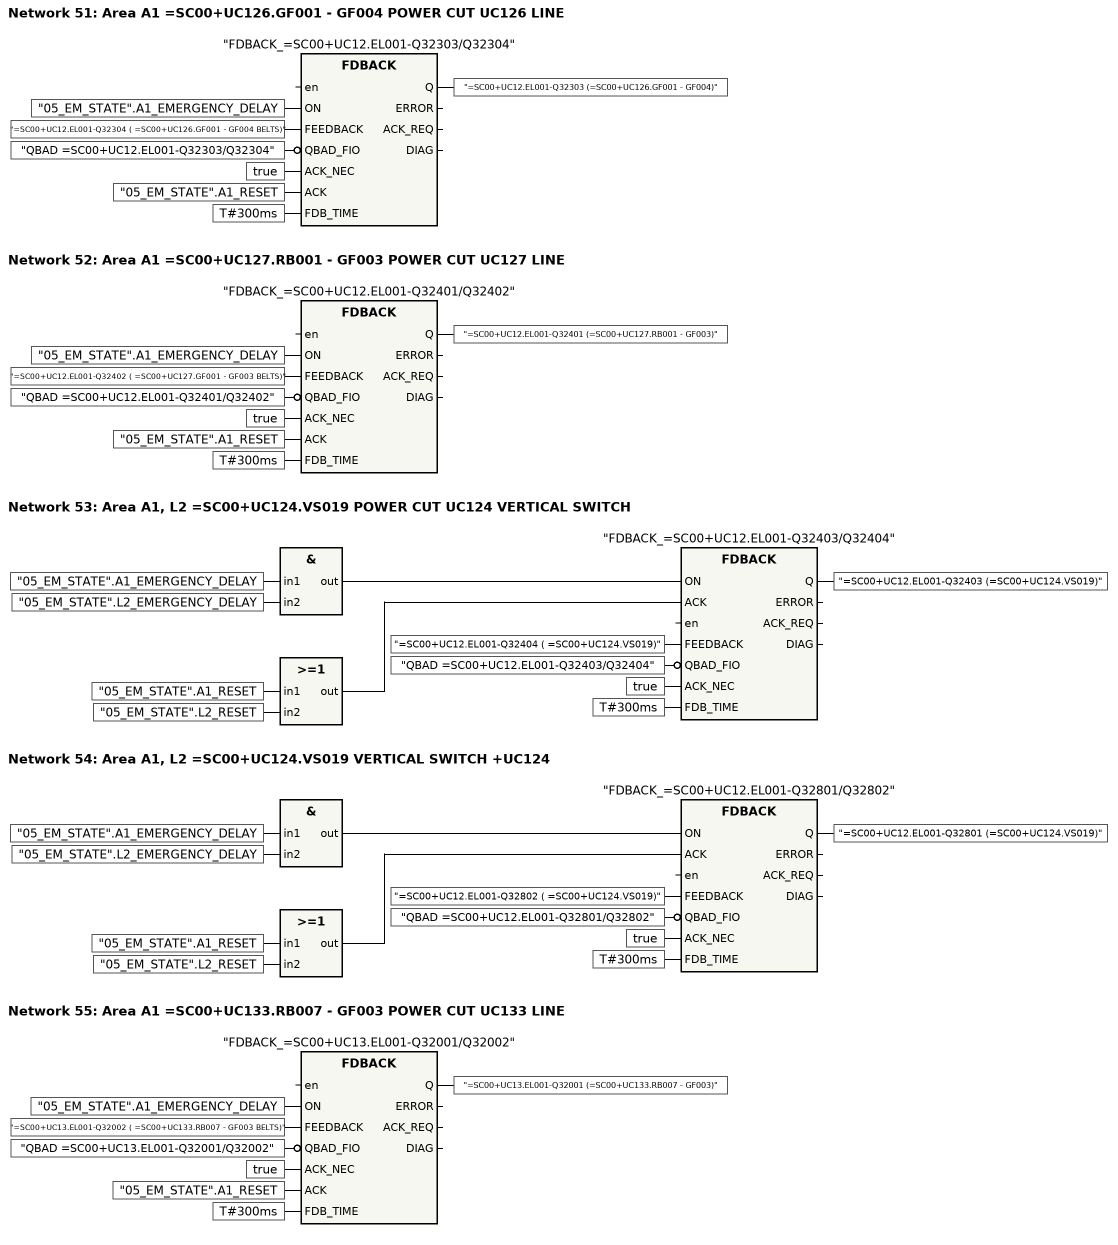
   "FDBACK_=SC00+UC12.EL001-Q32303/Q32304"(ON := "05_EM_STATE".A1_EMERGENCY_DELAY,   // FDBACK
                           FEEDBACK := "=SC00+UC12.EL001-Q32304 ( =SC00+UC126.GF001 - GF004 BELTS)",
                           QBAD_FIO := NOT "QBAD =SC00+UC12.EL001-Q32303/Q32304",
                           ACK_NEC := true,
                           ACK := "05_EM_STATE".A1_RESET,
                           FDB_TIME := T#300ms,
                           Q => "=SC00+UC12.EL001-Q32303 (=SC00+UC126.GF001 - GF004)");
END_REGION

REGION Network 52: Area A1 =SC00+UC127.RB001 - GF003 POWER CUT UC127 LINE
   "FDBACK_=SC00+UC12.EL001-Q32401/Q32402"(ON := "05_EM_STATE".A1_EMERGENCY_DELAY,   // FDBACK
                           FEEDBACK := "=SC00+UC12.EL001-Q32402 ( =SC00+UC127.GF001 - GF003 BELTS)",
                           QBAD_FIO := NOT "QBAD =SC00+UC12.EL001-Q32401/Q32402",
                           ACK_NEC := true,
                           ACK := "05_EM_STATE".A1_RESET,
                           FDB_TIME := T#300ms,
                           Q => "=SC00+UC12.EL001-Q32401 (=SC00+UC127.RB001 - GF003)");
END_REGION

REGION Network 53: Area A1, L2 =SC00+UC124.VS019 POWER CUT UC124 VERTICAL SWITCH
   "FDBACK_=SC00+UC12.EL001-Q32403/Q32404"(ON := "05_EM_STATE".A1_EMERGENCY_DELAY AND "05_EM_STATE".L2_EMERGENCY_DELAY,   // FDBACK
                           ACK := "05_EM_STATE".A1_RESET OR "05_EM_STATE".L2_RESET,
                           FEEDBACK := "=SC00+UC12.EL001-Q32404 ( =SC00+UC124.VS019)",
                           QBAD_FIO := NOT "QBAD =SC00+UC12.EL001-Q32403/Q32404",
                           ACK_NEC := true,
                           FDB_TIME := T#300ms,
                           Q => "=SC00+UC12.EL001-Q32403 (=SC00+UC124.VS019)");
END_REGION

REGION Network 54: Area A1, L2 =SC00+UC124.VS019 VERTICAL SWITCH +UC124
   "FDBACK_=SC00+UC12.EL001-Q32801/Q32802"(ON := "05_EM_STATE".A1_EMERGENCY_DELAY AND "05_EM_STATE".L2_EMERGENCY_DELAY,   // FDBACK
                           ACK := "05_EM_STATE".A1_RESET OR "05_EM_STATE".L2_RESET,
                           FEEDBACK := "=SC00+UC12.EL001-Q32802 ( =SC00+UC124.VS019)",
                           QBAD_FIO := NOT "QBAD =SC00+UC12.EL001-Q32801/Q32802",
                           ACK_NEC := true,
                           FDB_TIME := T#300ms,
                           Q => "=SC00+UC12.EL001-Q32801 (=SC00+UC124.VS019)");
END_REGION

REGION Network 55: Area A1 =SC00+UC133.RB007 - GF003 POWER CUT UC133 LINE
   "FDBACK_=SC00+UC13.EL001-Q32001/Q32002"(ON := "05_EM_STATE".A1_EMERGENCY_DELAY,   // FDBACK
                           FEEDBACK := "=SC00+UC13.EL001-Q32002 ( =SC00+UC133.RB007 - GF003 BELTS)",
                           QBAD_FIO := NOT "QBAD =SC00+UC13.EL001-Q32001/Q32002",
                           ACK_NEC := true,
                           ACK := "05_EM_STATE".A1_RESET,
                           FDB_TIME := T#300ms,
                           Q => "=SC00+UC13.EL001-Q32001 (=SC00+UC133.RB007 - GF003)");
END_REGION

REGION Network 56: Area A1 =SC00+UC132.RB007 - GF003 POWER CUT UC132 LINE
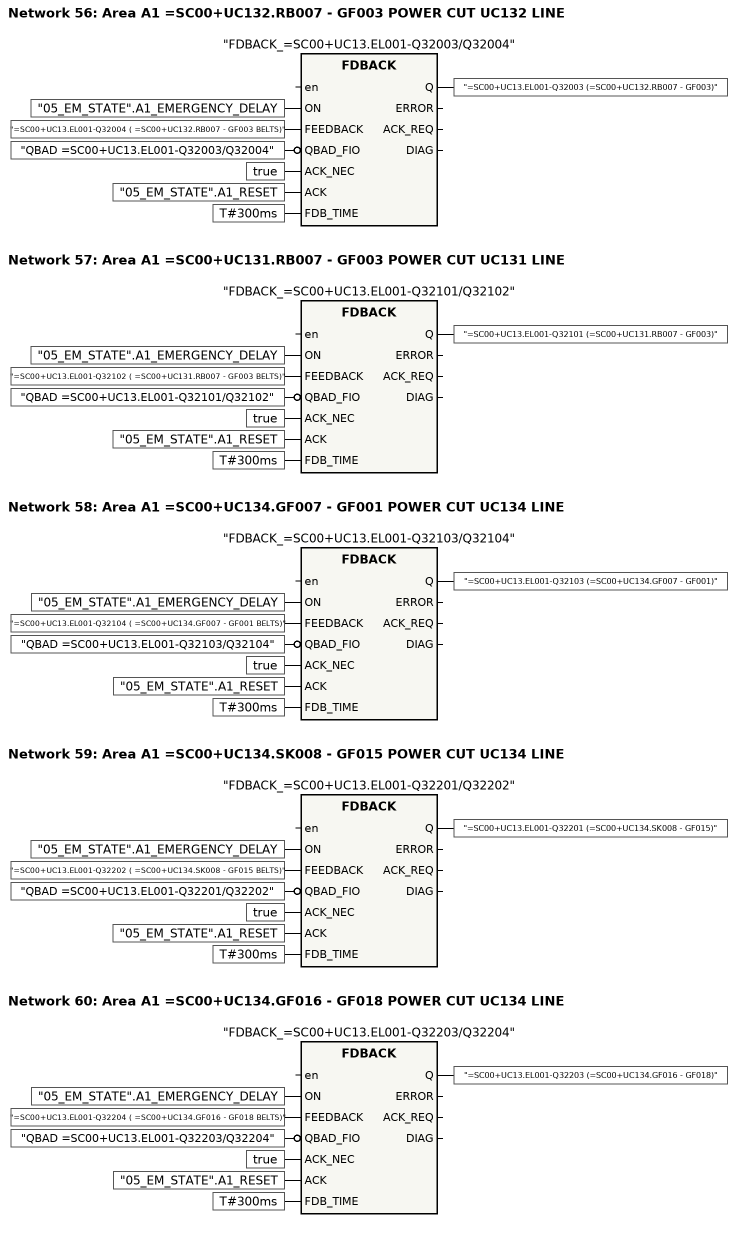
   "FDBACK_=SC00+UC13.EL001-Q32003/Q32004"(ON := "05_EM_STATE".A1_EMERGENCY_DELAY,   // FDBACK
                           FEEDBACK := "=SC00+UC13.EL001-Q32004 ( =SC00+UC132.RB007 - GF003 BELTS)",
                           QBAD_FIO := NOT "QBAD =SC00+UC13.EL001-Q32003/Q32004",
                           ACK_NEC := true,
                           ACK := "05_EM_STATE".A1_RESET,
                           FDB_TIME := T#300ms,
                           Q => "=SC00+UC13.EL001-Q32003 (=SC00+UC132.RB007 - GF003)");
END_REGION

REGION Network 57: Area A1 =SC00+UC131.RB007 - GF003 POWER CUT UC131 LINE
   "FDBACK_=SC00+UC13.EL001-Q32101/Q32102"(ON := "05_EM_STATE".A1_EMERGENCY_DELAY,   // FDBACK
                           FEEDBACK := "=SC00+UC13.EL001-Q32102 ( =SC00+UC131.RB007 - GF003 BELTS)",
                           QBAD_FIO := NOT "QBAD =SC00+UC13.EL001-Q32101/Q32102",
                           ACK_NEC := true,
                           ACK := "05_EM_STATE".A1_RESET,
                           FDB_TIME := T#300ms,
                           Q => "=SC00+UC13.EL001-Q32101 (=SC00+UC131.RB007 - GF003)");
END_REGION

REGION Network 58: Area A1 =SC00+UC134.GF007 - GF001 POWER CUT UC134 LINE
   "FDBACK_=SC00+UC13.EL001-Q32103/Q32104"(ON := "05_EM_STATE".A1_EMERGENCY_DELAY,   // FDBACK
                           FEEDBACK := "=SC00+UC13.EL001-Q32104 ( =SC00+UC134.GF007 - GF001 BELTS)",
                           QBAD_FIO := NOT "QBAD =SC00+UC13.EL001-Q32103/Q32104",
                           ACK_NEC := true,
                           ACK := "05_EM_STATE".A1_RESET,
                           FDB_TIME := T#300ms,
                           Q => "=SC00+UC13.EL001-Q32103 (=SC00+UC134.GF007 - GF001)");
END_REGION

REGION Network 59: Area A1 =SC00+UC134.SK008 - GF015 POWER CUT UC134 LINE
   "FDBACK_=SC00+UC13.EL001-Q32201/Q32202"(ON := "05_EM_STATE".A1_EMERGENCY_DELAY,   // FDBACK
                           FEEDBACK := "=SC00+UC13.EL001-Q32202 ( =SC00+UC134.SK008 - GF015 BELTS)",
                           QBAD_FIO := NOT "QBAD =SC00+UC13.EL001-Q32201/Q32202",
                           ACK_NEC := true,
                           ACK := "05_EM_STATE".A1_RESET,
                           FDB_TIME := T#300ms,
                           Q => "=SC00+UC13.EL001-Q32201 (=SC00+UC134.SK008 - GF015)");
END_REGION

REGION Network 60: Area A1 =SC00+UC134.GF016 - GF018 POWER CUT UC134 LINE
   "FDBACK_=SC00+UC13.EL001-Q32203/Q32204"(ON := "05_EM_STATE".A1_EMERGENCY_DELAY,   // FDBACK
                           FEEDBACK := "=SC00+UC13.EL001-Q32204 ( =SC00+UC134.GF016 - GF018 BELTS)",
                           QBAD_FIO := NOT "QBAD =SC00+UC13.EL001-Q32203/Q32204",
                           ACK_NEC := true,
                           ACK := "05_EM_STATE".A1_RESET,
                           FDB_TIME := T#300ms,
                           Q => "=SC00+UC13.EL001-Q32203 (=SC00+UC134.GF016 - GF018)");
END_REGION

REGION Network 61: Area A1 =SC00+UC135.GF001 - GF004 POWER CUT UC135 LINE
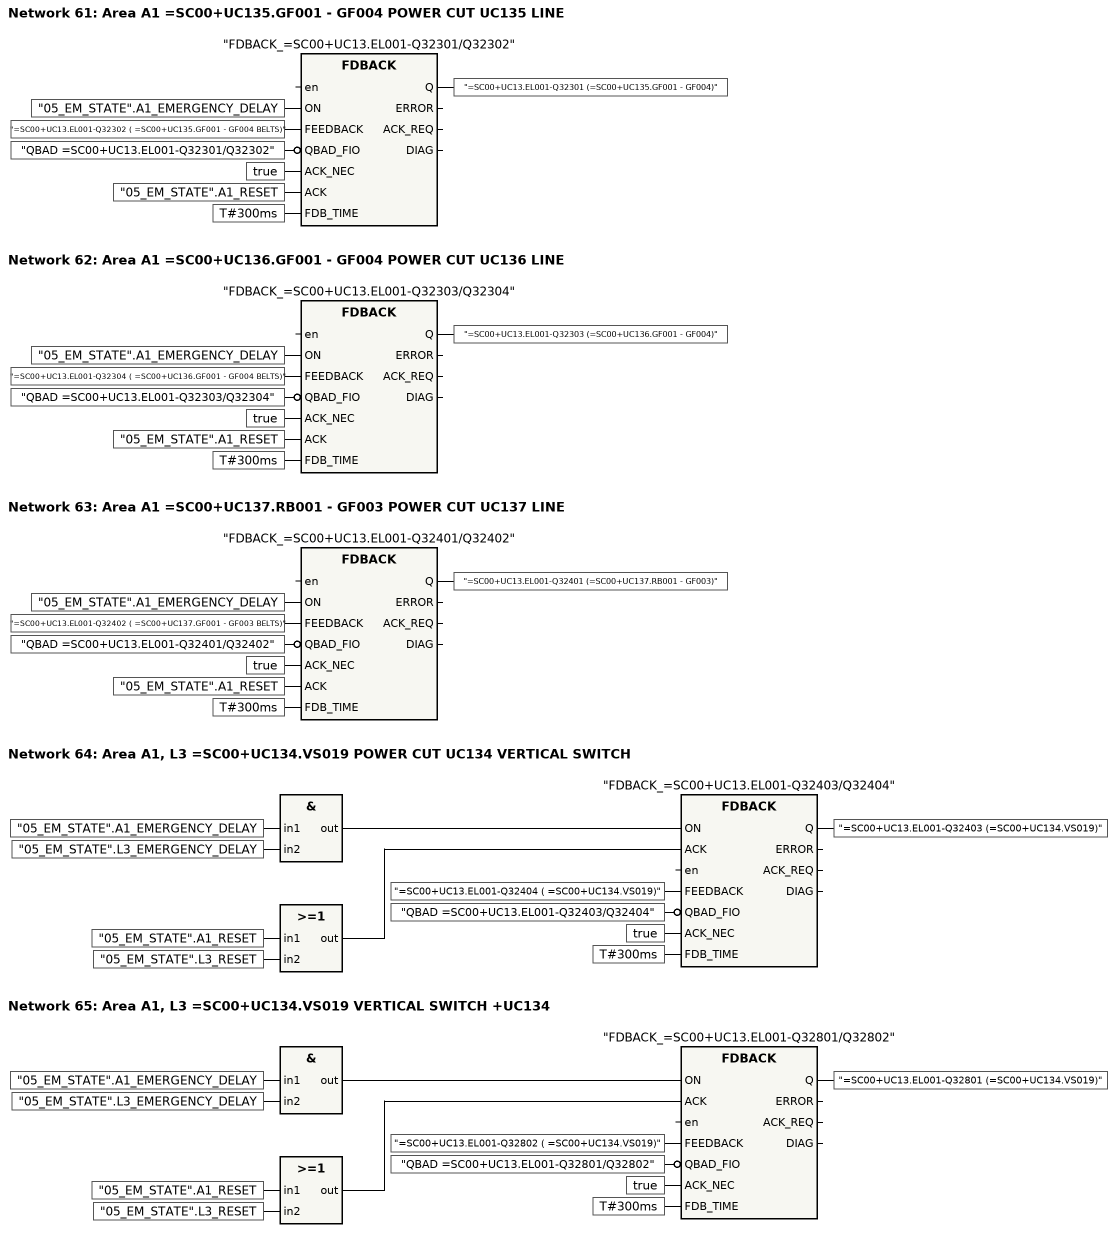
   "FDBACK_=SC00+UC13.EL001-Q32301/Q32302"(ON := "05_EM_STATE".A1_EMERGENCY_DELAY,   // FDBACK
                           FEEDBACK := "=SC00+UC13.EL001-Q32302 ( =SC00+UC135.GF001 - GF004 BELTS)",
                           QBAD_FIO := NOT "QBAD =SC00+UC13.EL001-Q32301/Q32302",
                           ACK_NEC := true,
                           ACK := "05_EM_STATE".A1_RESET,
                           FDB_TIME := T#300ms,
                           Q => "=SC00+UC13.EL001-Q32301 (=SC00+UC135.GF001 - GF004)");
END_REGION

REGION Network 62: Area A1 =SC00+UC136.GF001 - GF004 POWER CUT UC136 LINE
   "FDBACK_=SC00+UC13.EL001-Q32303/Q32304"(ON := "05_EM_STATE".A1_EMERGENCY_DELAY,   // FDBACK
                           FEEDBACK := "=SC00+UC13.EL001-Q32304 ( =SC00+UC136.GF001 - GF004 BELTS)",
                           QBAD_FIO := NOT "QBAD =SC00+UC13.EL001-Q32303/Q32304",
                           ACK_NEC := true,
                           ACK := "05_EM_STATE".A1_RESET,
                           FDB_TIME := T#300ms,
                           Q => "=SC00+UC13.EL001-Q32303 (=SC00+UC136.GF001 - GF004)");
END_REGION

REGION Network 63: Area A1 =SC00+UC137.RB001 - GF003 POWER CUT UC137 LINE
   "FDBACK_=SC00+UC13.EL001-Q32401/Q32402"(ON := "05_EM_STATE".A1_EMERGENCY_DELAY,   // FDBACK
                           FEEDBACK := "=SC00+UC13.EL001-Q32402 ( =SC00+UC137.GF001 - GF003 BELTS)",
                           QBAD_FIO := NOT "QBAD =SC00+UC13.EL001-Q32401/Q32402",
                           ACK_NEC := true,
                           ACK := "05_EM_STATE".A1_RESET,
                           FDB_TIME := T#300ms,
                           Q => "=SC00+UC13.EL001-Q32401 (=SC00+UC137.RB001 - GF003)");
END_REGION

REGION Network 64: Area A1, L3 =SC00+UC134.VS019 POWER CUT UC134 VERTICAL SWITCH
   "FDBACK_=SC00+UC13.EL001-Q32403/Q32404"(ON := "05_EM_STATE".A1_EMERGENCY_DELAY AND "05_EM_STATE".L3_EMERGENCY_DELAY,   // FDBACK
                           ACK := "05_EM_STATE".A1_RESET OR "05_EM_STATE".L3_RESET,
                           FEEDBACK := "=SC00+UC13.EL001-Q32404 ( =SC00+UC134.VS019)",
                           QBAD_FIO := NOT "QBAD =SC00+UC13.EL001-Q32403/Q32404",
                           ACK_NEC := true,
                           FDB_TIME := T#300ms,
                           Q => "=SC00+UC13.EL001-Q32403 (=SC00+UC134.VS019)");
END_REGION

REGION Network 65: Area A1, L3 =SC00+UC134.VS019 VERTICAL SWITCH +UC134
   "FDBACK_=SC00+UC13.EL001-Q32801/Q32802"(ON := "05_EM_STATE".A1_EMERGENCY_DELAY AND "05_EM_STATE".L3_EMERGENCY_DELAY,   // FDBACK
                           ACK := "05_EM_STATE".A1_RESET OR "05_EM_STATE".L3_RESET,
                           FEEDBACK := "=SC00+UC13.EL001-Q32802 ( =SC00+UC134.VS019)",
                           QBAD_FIO := NOT "QBAD =SC00+UC13.EL001-Q32801/Q32802",
                           ACK_NEC := true,
                           FDB_TIME := T#300ms,
                           Q => "=SC00+UC13.EL001-Q32801 (=SC00+UC134.VS019)");
END_REGION

REGION Network 66: Area A1 =SC00+UC143.RB007 - GF003 POWER CUT UC143 LINE
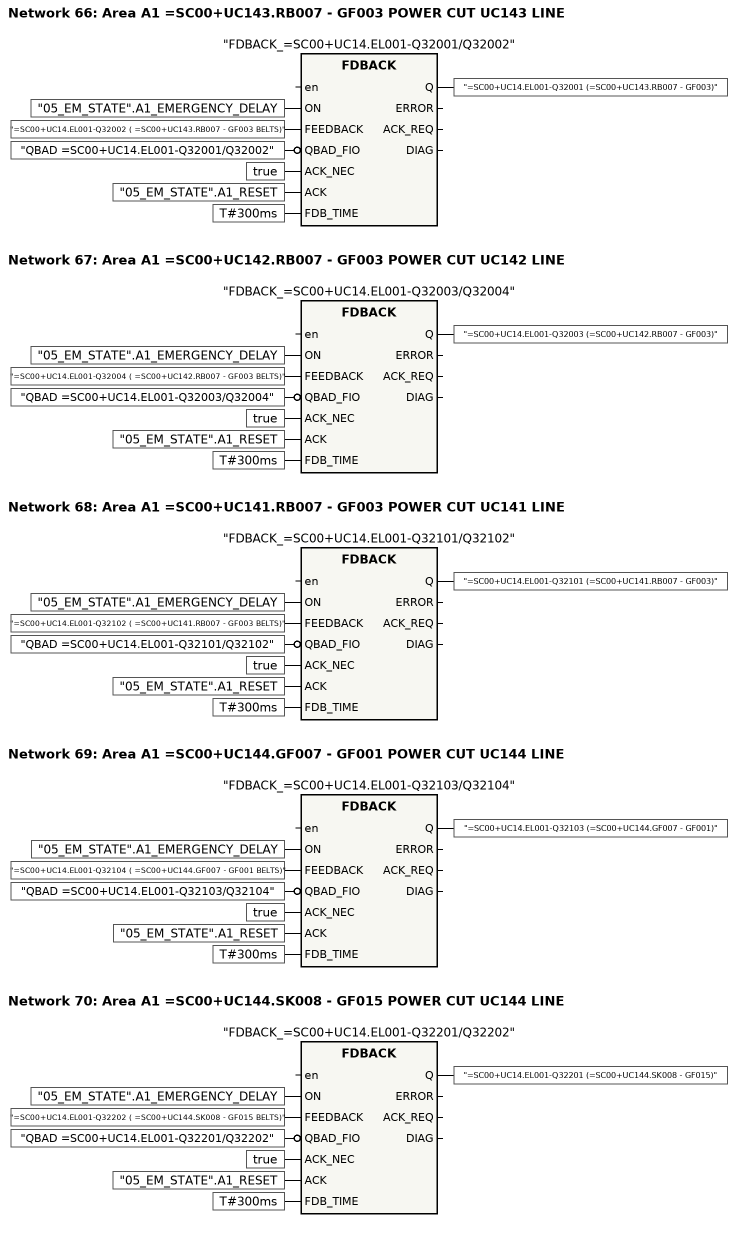
   "FDBACK_=SC00+UC14.EL001-Q32001/Q32002"(ON := "05_EM_STATE".A1_EMERGENCY_DELAY,   // FDBACK
                           FEEDBACK := "=SC00+UC14.EL001-Q32002 ( =SC00+UC143.RB007 - GF003 BELTS)",
                           QBAD_FIO := NOT "QBAD =SC00+UC14.EL001-Q32001/Q32002",
                           ACK_NEC := true,
                           ACK := "05_EM_STATE".A1_RESET,
                           FDB_TIME := T#300ms,
                           Q => "=SC00+UC14.EL001-Q32001 (=SC00+UC143.RB007 - GF003)");
END_REGION

REGION Network 67: Area A1 =SC00+UC142.RB007 - GF003 POWER CUT UC142 LINE
   "FDBACK_=SC00+UC14.EL001-Q32003/Q32004"(ON := "05_EM_STATE".A1_EMERGENCY_DELAY,   // FDBACK
                           FEEDBACK := "=SC00+UC14.EL001-Q32004 ( =SC00+UC142.RB007 - GF003 BELTS)",
                           QBAD_FIO := NOT "QBAD =SC00+UC14.EL001-Q32003/Q32004",
                           ACK_NEC := true,
                           ACK := "05_EM_STATE".A1_RESET,
                           FDB_TIME := T#300ms,
                           Q => "=SC00+UC14.EL001-Q32003 (=SC00+UC142.RB007 - GF003)");
END_REGION

REGION Network 68: Area A1 =SC00+UC141.RB007 - GF003 POWER CUT UC141 LINE
   "FDBACK_=SC00+UC14.EL001-Q32101/Q32102"(ON := "05_EM_STATE".A1_EMERGENCY_DELAY,   // FDBACK
                           FEEDBACK := "=SC00+UC14.EL001-Q32102 ( =SC00+UC141.RB007 - GF003 BELTS)",
                           QBAD_FIO := NOT "QBAD =SC00+UC14.EL001-Q32101/Q32102",
                           ACK_NEC := true,
                           ACK := "05_EM_STATE".A1_RESET,
                           FDB_TIME := T#300ms,
                           Q => "=SC00+UC14.EL001-Q32101 (=SC00+UC141.RB007 - GF003)");
END_REGION

REGION Network 69: Area A1 =SC00+UC144.GF007 - GF001 POWER CUT UC144 LINE
   "FDBACK_=SC00+UC14.EL001-Q32103/Q32104"(ON := "05_EM_STATE".A1_EMERGENCY_DELAY,   // FDBACK
                           FEEDBACK := "=SC00+UC14.EL001-Q32104 ( =SC00+UC144.GF007 - GF001 BELTS)",
                           QBAD_FIO := NOT "QBAD =SC00+UC14.EL001-Q32103/Q32104",
                           ACK_NEC := true,
                           ACK := "05_EM_STATE".A1_RESET,
                           FDB_TIME := T#300ms,
                           Q => "=SC00+UC14.EL001-Q32103 (=SC00+UC144.GF007 - GF001)");
END_REGION

REGION Network 70: Area A1 =SC00+UC144.SK008 - GF015 POWER CUT UC144 LINE
   "FDBACK_=SC00+UC14.EL001-Q32201/Q32202"(ON := "05_EM_STATE".A1_EMERGENCY_DELAY,   // FDBACK
                           FEEDBACK := "=SC00+UC14.EL001-Q32202 ( =SC00+UC144.SK008 - GF015 BELTS)",
                           QBAD_FIO := NOT "QBAD =SC00+UC14.EL001-Q32201/Q32202",
                           ACK_NEC := true,
                           ACK := "05_EM_STATE".A1_RESET,
                           FDB_TIME := T#300ms,
                           Q => "=SC00+UC14.EL001-Q32201 (=SC00+UC144.SK008 - GF015)");
END_REGION

REGION Network 71: Area A1 =SC00+UC144.GF016 - GF018 POWER CUT UC144 LINE
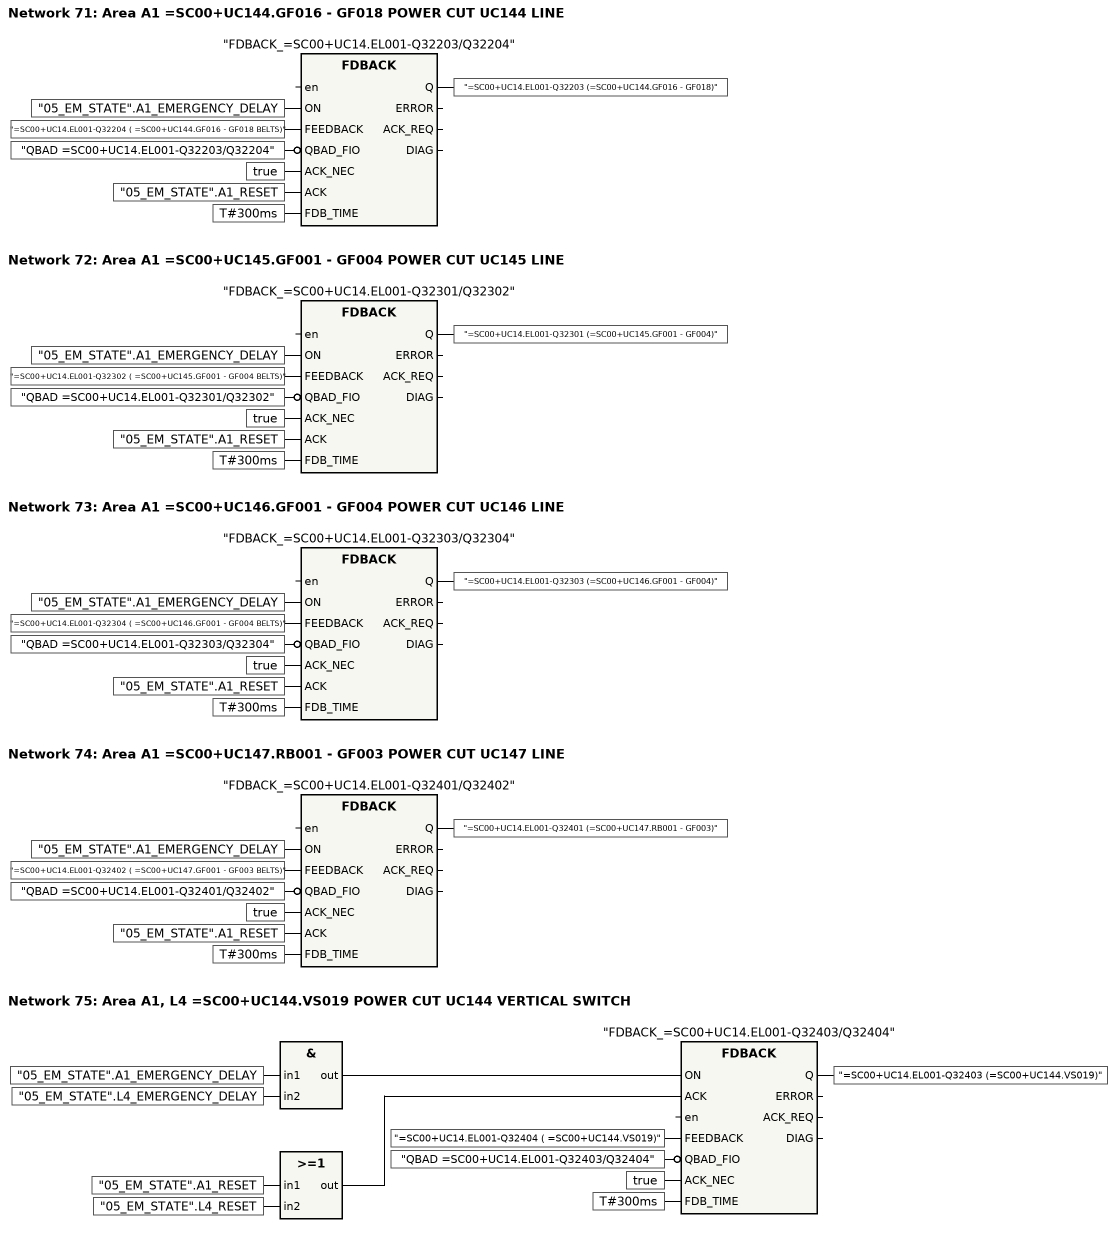
   "FDBACK_=SC00+UC14.EL001-Q32203/Q32204"(ON := "05_EM_STATE".A1_EMERGENCY_DELAY,   // FDBACK
                           FEEDBACK := "=SC00+UC14.EL001-Q32204 ( =SC00+UC144.GF016 - GF018 BELTS)",
                           QBAD_FIO := NOT "QBAD =SC00+UC14.EL001-Q32203/Q32204",
                           ACK_NEC := true,
                           ACK := "05_EM_STATE".A1_RESET,
                           FDB_TIME := T#300ms,
                           Q => "=SC00+UC14.EL001-Q32203 (=SC00+UC144.GF016 - GF018)");
END_REGION

REGION Network 72: Area A1 =SC00+UC145.GF001 - GF004 POWER CUT UC145 LINE
   "FDBACK_=SC00+UC14.EL001-Q32301/Q32302"(ON := "05_EM_STATE".A1_EMERGENCY_DELAY,   // FDBACK
                           FEEDBACK := "=SC00+UC14.EL001-Q32302 ( =SC00+UC145.GF001 - GF004 BELTS)",
                           QBAD_FIO := NOT "QBAD =SC00+UC14.EL001-Q32301/Q32302",
                           ACK_NEC := true,
                           ACK := "05_EM_STATE".A1_RESET,
                           FDB_TIME := T#300ms,
                           Q => "=SC00+UC14.EL001-Q32301 (=SC00+UC145.GF001 - GF004)");
END_REGION

REGION Network 73: Area A1 =SC00+UC146.GF001 - GF004 POWER CUT UC146 LINE
   "FDBACK_=SC00+UC14.EL001-Q32303/Q32304"(ON := "05_EM_STATE".A1_EMERGENCY_DELAY,   // FDBACK
                           FEEDBACK := "=SC00+UC14.EL001-Q32304 ( =SC00+UC146.GF001 - GF004 BELTS)",
                           QBAD_FIO := NOT "QBAD =SC00+UC14.EL001-Q32303/Q32304",
                           ACK_NEC := true,
                           ACK := "05_EM_STATE".A1_RESET,
                           FDB_TIME := T#300ms,
                           Q => "=SC00+UC14.EL001-Q32303 (=SC00+UC146.GF001 - GF004)");
END_REGION

REGION Network 74: Area A1 =SC00+UC147.RB001 - GF003 POWER CUT UC147 LINE
   "FDBACK_=SC00+UC14.EL001-Q32401/Q32402"(ON := "05_EM_STATE".A1_EMERGENCY_DELAY,   // FDBACK
                           FEEDBACK := "=SC00+UC14.EL001-Q32402 ( =SC00+UC147.GF001 - GF003 BELTS)",
                           QBAD_FIO := NOT "QBAD =SC00+UC14.EL001-Q32401/Q32402",
                           ACK_NEC := true,
                           ACK := "05_EM_STATE".A1_RESET,
                           FDB_TIME := T#300ms,
                           Q => "=SC00+UC14.EL001-Q32401 (=SC00+UC147.RB001 - GF003)");
END_REGION

REGION Network 75: Area A1, L4 =SC00+UC144.VS019 POWER CUT UC144 VERTICAL SWITCH
   "FDBACK_=SC00+UC14.EL001-Q32403/Q32404"(ON := "05_EM_STATE".A1_EMERGENCY_DELAY AND "05_EM_STATE".L4_EMERGENCY_DELAY,   // FDBACK
                           ACK := "05_EM_STATE".A1_RESET OR "05_EM_STATE".L4_RESET,
                           FEEDBACK := "=SC00+UC14.EL001-Q32404 ( =SC00+UC144.VS019)",
                           QBAD_FIO := NOT "QBAD =SC00+UC14.EL001-Q32403/Q32404",
                           ACK_NEC := true,
                           FDB_TIME := T#300ms,
                           Q => "=SC00+UC14.EL001-Q32403 (=SC00+UC144.VS019)");
END_REGION

REGION Network 76: Area A1, L4 =SC00+UC144.VS019 VERTICAL SWITCH +UC144
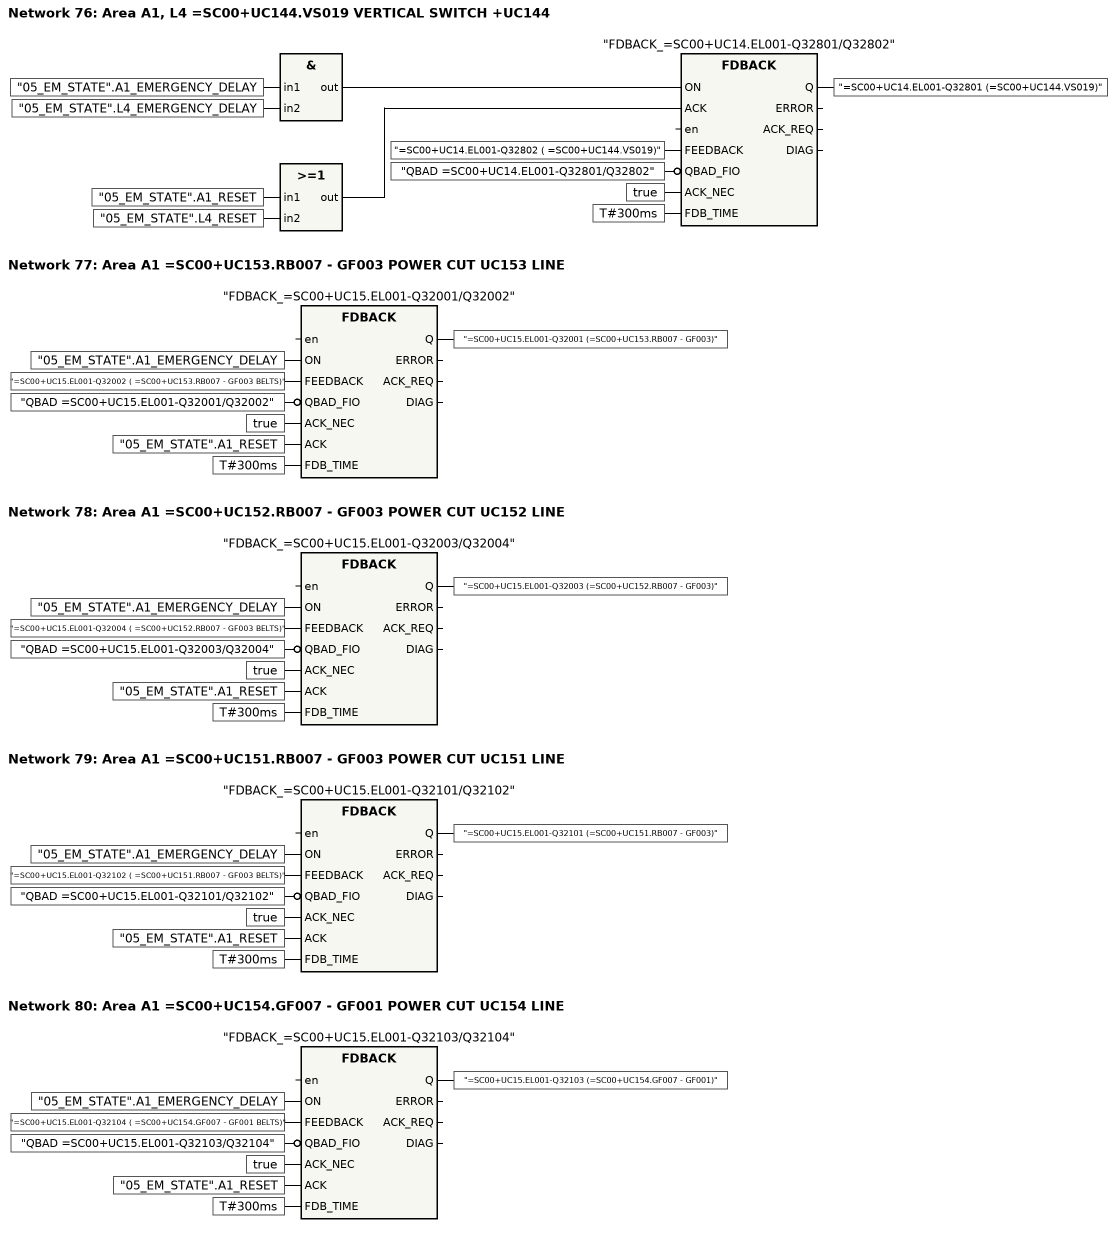
   "FDBACK_=SC00+UC14.EL001-Q32801/Q32802"(ON := "05_EM_STATE".A1_EMERGENCY_DELAY AND "05_EM_STATE".L4_EMERGENCY_DELAY,   // FDBACK
                           ACK := "05_EM_STATE".A1_RESET OR "05_EM_STATE".L4_RESET,
                           FEEDBACK := "=SC00+UC14.EL001-Q32802 ( =SC00+UC144.VS019)",
                           QBAD_FIO := NOT "QBAD =SC00+UC14.EL001-Q32801/Q32802",
                           ACK_NEC := true,
                           FDB_TIME := T#300ms,
                           Q => "=SC00+UC14.EL001-Q32801 (=SC00+UC144.VS019)");
END_REGION

REGION Network 77: Area A1 =SC00+UC153.RB007 - GF003 POWER CUT UC153 LINE
   "FDBACK_=SC00+UC15.EL001-Q32001/Q32002"(ON := "05_EM_STATE".A1_EMERGENCY_DELAY,   // FDBACK
                           FEEDBACK := "=SC00+UC15.EL001-Q32002 ( =SC00+UC153.RB007 - GF003 BELTS)",
                           QBAD_FIO := NOT "QBAD =SC00+UC15.EL001-Q32001/Q32002",
                           ACK_NEC := true,
                           ACK := "05_EM_STATE".A1_RESET,
                           FDB_TIME := T#300ms,
                           Q => "=SC00+UC15.EL001-Q32001 (=SC00+UC153.RB007 - GF003)");
END_REGION

REGION Network 78: Area A1 =SC00+UC152.RB007 - GF003 POWER CUT UC152 LINE
   "FDBACK_=SC00+UC15.EL001-Q32003/Q32004"(ON := "05_EM_STATE".A1_EMERGENCY_DELAY,   // FDBACK
                           FEEDBACK := "=SC00+UC15.EL001-Q32004 ( =SC00+UC152.RB007 - GF003 BELTS)",
                           QBAD_FIO := NOT "QBAD =SC00+UC15.EL001-Q32003/Q32004",
                           ACK_NEC := true,
                           ACK := "05_EM_STATE".A1_RESET,
                           FDB_TIME := T#300ms,
                           Q => "=SC00+UC15.EL001-Q32003 (=SC00+UC152.RB007 - GF003)");
END_REGION

REGION Network 79: Area A1 =SC00+UC151.RB007 - GF003 POWER CUT UC151 LINE
   "FDBACK_=SC00+UC15.EL001-Q32101/Q32102"(ON := "05_EM_STATE".A1_EMERGENCY_DELAY,   // FDBACK
                           FEEDBACK := "=SC00+UC15.EL001-Q32102 ( =SC00+UC151.RB007 - GF003 BELTS)",
                           QBAD_FIO := NOT "QBAD =SC00+UC15.EL001-Q32101/Q32102",
                           ACK_NEC := true,
                           ACK := "05_EM_STATE".A1_RESET,
                           FDB_TIME := T#300ms,
                           Q => "=SC00+UC15.EL001-Q32101 (=SC00+UC151.RB007 - GF003)");
END_REGION

REGION Network 80: Area A1 =SC00+UC154.GF007 - GF001 POWER CUT UC154 LINE
   "FDBACK_=SC00+UC15.EL001-Q32103/Q32104"(ON := "05_EM_STATE".A1_EMERGENCY_DELAY,   // FDBACK
                           FEEDBACK := "=SC00+UC15.EL001-Q32104 ( =SC00+UC154.GF007 - GF001 BELTS)",
                           QBAD_FIO := NOT "QBAD =SC00+UC15.EL001-Q32103/Q32104",
                           ACK_NEC := true,
                           ACK := "05_EM_STATE".A1_RESET,
                           FDB_TIME := T#300ms,
                           Q => "=SC00+UC15.EL001-Q32103 (=SC00+UC154.GF007 - GF001)");
END_REGION

REGION Network 81: Area A1 =SC00+UC154.SK008 - GF015 POWER CUT UC154 LINE
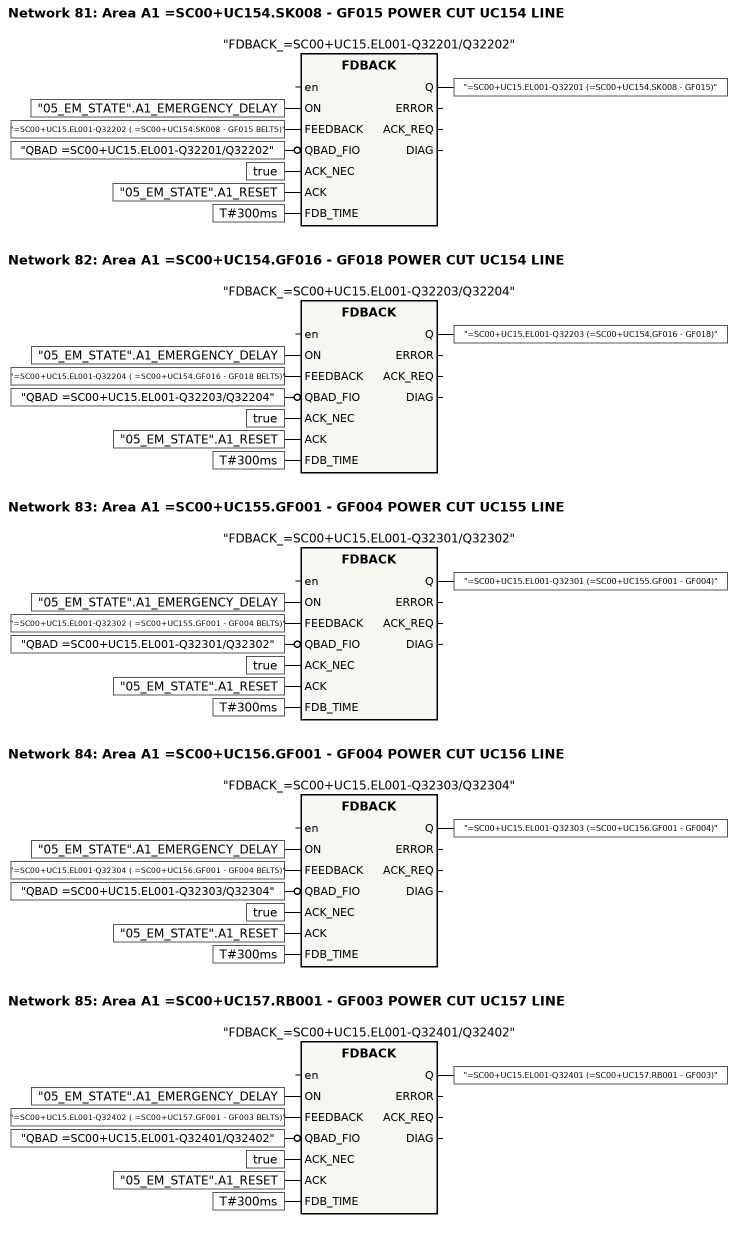
   "FDBACK_=SC00+UC15.EL001-Q32201/Q32202"(ON := "05_EM_STATE".A1_EMERGENCY_DELAY,   // FDBACK
                           FEEDBACK := "=SC00+UC15.EL001-Q32202 ( =SC00+UC154.SK008 - GF015 BELTS)",
                           QBAD_FIO := NOT "QBAD =SC00+UC15.EL001-Q32201/Q32202",
                           ACK_NEC := true,
                           ACK := "05_EM_STATE".A1_RESET,
                           FDB_TIME := T#300ms,
                           Q => "=SC00+UC15.EL001-Q32201 (=SC00+UC154.SK008 - GF015)");
END_REGION

REGION Network 82: Area A1 =SC00+UC154.GF016 - GF018 POWER CUT UC154 LINE
   "FDBACK_=SC00+UC15.EL001-Q32203/Q32204"(ON := "05_EM_STATE".A1_EMERGENCY_DELAY,   // FDBACK
                           FEEDBACK := "=SC00+UC15.EL001-Q32204 ( =SC00+UC154.GF016 - GF018 BELTS)",
                           QBAD_FIO := NOT "QBAD =SC00+UC15.EL001-Q32203/Q32204",
                           ACK_NEC := true,
                           ACK := "05_EM_STATE".A1_RESET,
                           FDB_TIME := T#300ms,
                           Q => "=SC00+UC15.EL001-Q32203 (=SC00+UC154.GF016 - GF018)");
END_REGION

REGION Network 83: Area A1 =SC00+UC155.GF001 - GF004 POWER CUT UC155 LINE
   "FDBACK_=SC00+UC15.EL001-Q32301/Q32302"(ON := "05_EM_STATE".A1_EMERGENCY_DELAY,   // FDBACK
                           FEEDBACK := "=SC00+UC15.EL001-Q32302 ( =SC00+UC155.GF001 - GF004 BELTS)",
                           QBAD_FIO := NOT "QBAD =SC00+UC15.EL001-Q32301/Q32302",
                           ACK_NEC := true,
                           ACK := "05_EM_STATE".A1_RESET,
                           FDB_TIME := T#300ms,
                           Q => "=SC00+UC15.EL001-Q32301 (=SC00+UC155.GF001 - GF004)");
END_REGION

REGION Network 84: Area A1 =SC00+UC156.GF001 - GF004 POWER CUT UC156 LINE
   "FDBACK_=SC00+UC15.EL001-Q32303/Q32304"(ON := "05_EM_STATE".A1_EMERGENCY_DELAY,   // FDBACK
                           FEEDBACK := "=SC00+UC15.EL001-Q32304 ( =SC00+UC156.GF001 - GF004 BELTS)",
                           QBAD_FIO := NOT "QBAD =SC00+UC15.EL001-Q32303/Q32304",
                           ACK_NEC := true,
                           ACK := "05_EM_STATE".A1_RESET,
                           FDB_TIME := T#300ms,
                           Q => "=SC00+UC15.EL001-Q32303 (=SC00+UC156.GF001 - GF004)");
END_REGION

REGION Network 85: Area A1 =SC00+UC157.RB001 - GF003 POWER CUT UC157 LINE
   "FDBACK_=SC00+UC15.EL001-Q32401/Q32402"(ON := "05_EM_STATE".A1_EMERGENCY_DELAY,   // FDBACK
                           FEEDBACK := "=SC00+UC15.EL001-Q32402 ( =SC00+UC157.GF001 - GF003 BELTS)",
                           QBAD_FIO := NOT "QBAD =SC00+UC15.EL001-Q32401/Q32402",
                           ACK_NEC := true,
                           ACK := "05_EM_STATE".A1_RESET,
                           FDB_TIME := T#300ms,
                           Q => "=SC00+UC15.EL001-Q32401 (=SC00+UC157.RB001 - GF003)");
END_REGION

REGION Network 86: Area A1, L5 =SC00+UC154.VS019 POWER CUT UC154 VERTICAL SWITCH
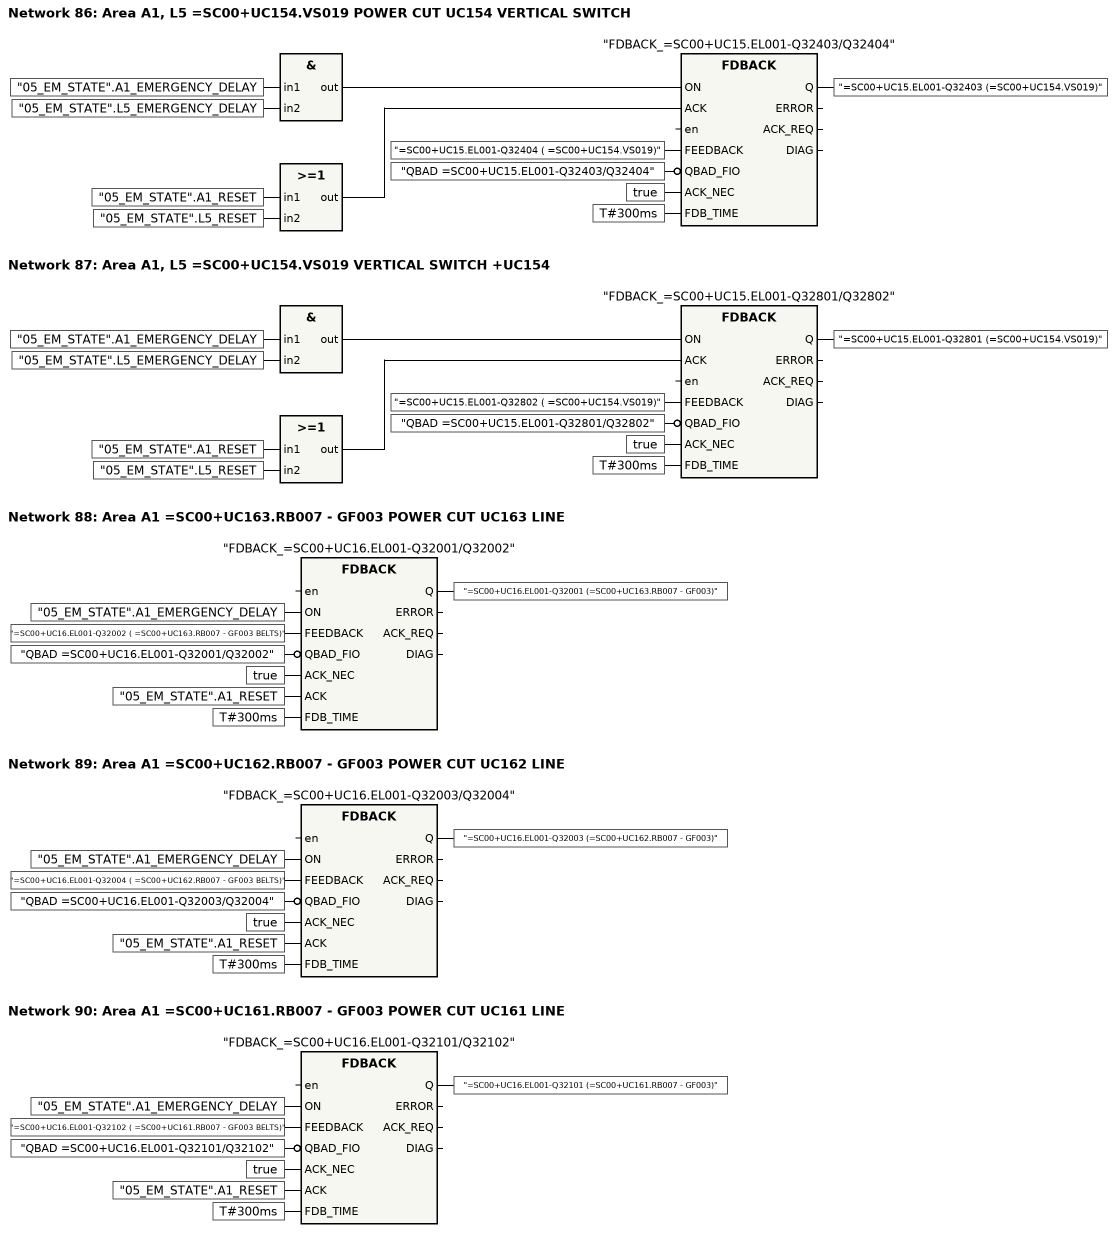
   "FDBACK_=SC00+UC15.EL001-Q32403/Q32404"(ON := "05_EM_STATE".A1_EMERGENCY_DELAY AND "05_EM_STATE".L5_EMERGENCY_DELAY,   // FDBACK
                           ACK := "05_EM_STATE".A1_RESET OR "05_EM_STATE".L5_RESET,
                           FEEDBACK := "=SC00+UC15.EL001-Q32404 ( =SC00+UC154.VS019)",
                           QBAD_FIO := NOT "QBAD =SC00+UC15.EL001-Q32403/Q32404",
                           ACK_NEC := true,
                           FDB_TIME := T#300ms,
                           Q => "=SC00+UC15.EL001-Q32403 (=SC00+UC154.VS019)");
END_REGION

REGION Network 87: Area A1, L5 =SC00+UC154.VS019 VERTICAL SWITCH +UC154
   "FDBACK_=SC00+UC15.EL001-Q32801/Q32802"(ON := "05_EM_STATE".A1_EMERGENCY_DELAY AND "05_EM_STATE".L5_EMERGENCY_DELAY,   // FDBACK
                           ACK := "05_EM_STATE".A1_RESET OR "05_EM_STATE".L5_RESET,
                           FEEDBACK := "=SC00+UC15.EL001-Q32802 ( =SC00+UC154.VS019)",
                           QBAD_FIO := NOT "QBAD =SC00+UC15.EL001-Q32801/Q32802",
                           ACK_NEC := true,
                           FDB_TIME := T#300ms,
                           Q => "=SC00+UC15.EL001-Q32801 (=SC00+UC154.VS019)");
END_REGION

REGION Network 88: Area A1 =SC00+UC163.RB007 - GF003 POWER CUT UC163 LINE
   "FDBACK_=SC00+UC16.EL001-Q32001/Q32002"(ON := "05_EM_STATE".A1_EMERGENCY_DELAY,   // FDBACK
                           FEEDBACK := "=SC00+UC16.EL001-Q32002 ( =SC00+UC163.RB007 - GF003 BELTS)",
                           QBAD_FIO := NOT "QBAD =SC00+UC16.EL001-Q32001/Q32002",
                           ACK_NEC := true,
                           ACK := "05_EM_STATE".A1_RESET,
                           FDB_TIME := T#300ms,
                           Q => "=SC00+UC16.EL001-Q32001 (=SC00+UC163.RB007 - GF003)");
END_REGION

REGION Network 89: Area A1 =SC00+UC162.RB007 - GF003 POWER CUT UC162 LINE
   "FDBACK_=SC00+UC16.EL001-Q32003/Q32004"(ON := "05_EM_STATE".A1_EMERGENCY_DELAY,   // FDBACK
                           FEEDBACK := "=SC00+UC16.EL001-Q32004 ( =SC00+UC162.RB007 - GF003 BELTS)",
                           QBAD_FIO := NOT "QBAD =SC00+UC16.EL001-Q32003/Q32004",
                           ACK_NEC := true,
                           ACK := "05_EM_STATE".A1_RESET,
                           FDB_TIME := T#300ms,
                           Q => "=SC00+UC16.EL001-Q32003 (=SC00+UC162.RB007 - GF003)");
END_REGION

REGION Network 90: Area A1 =SC00+UC161.RB007 - GF003 POWER CUT UC161 LINE
   "FDBACK_=SC00+UC16.EL001-Q32101/Q32102"(ON := "05_EM_STATE".A1_EMERGENCY_DELAY,   // FDBACK
                           FEEDBACK := "=SC00+UC16.EL001-Q32102 ( =SC00+UC161.RB007 - GF003 BELTS)",
                           QBAD_FIO := NOT "QBAD =SC00+UC16.EL001-Q32101/Q32102",
                           ACK_NEC := true,
                           ACK := "05_EM_STATE".A1_RESET,
                           FDB_TIME := T#300ms,
                           Q => "=SC00+UC16.EL001-Q32101 (=SC00+UC161.RB007 - GF003)");
END_REGION

REGION Network 91: Area A1 =SC00+UC164.GF007 - GF001 POWER CUT UC164 LINE
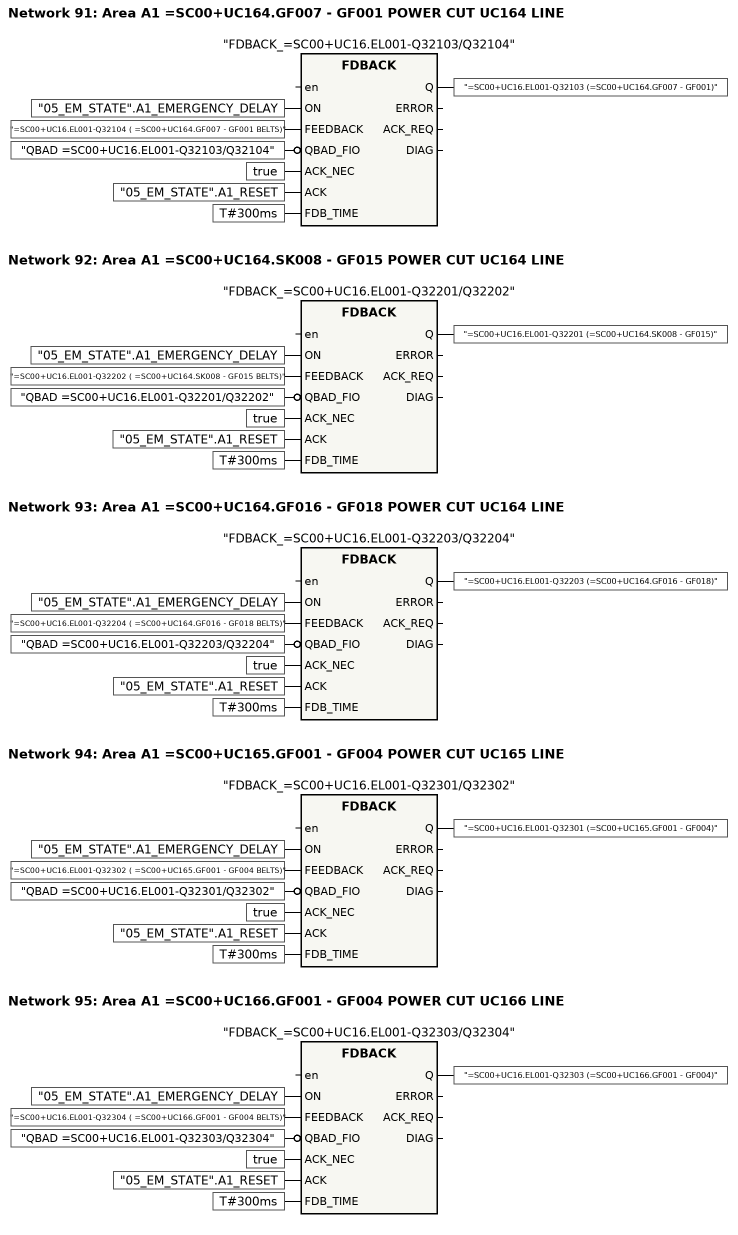
   "FDBACK_=SC00+UC16.EL001-Q32103/Q32104"(ON := "05_EM_STATE".A1_EMERGENCY_DELAY,   // FDBACK
                           FEEDBACK := "=SC00+UC16.EL001-Q32104 ( =SC00+UC164.GF007 - GF001 BELTS)",
                           QBAD_FIO := NOT "QBAD =SC00+UC16.EL001-Q32103/Q32104",
                           ACK_NEC := true,
                           ACK := "05_EM_STATE".A1_RESET,
                           FDB_TIME := T#300ms,
                           Q => "=SC00+UC16.EL001-Q32103 (=SC00+UC164.GF007 - GF001)");
END_REGION

REGION Network 92: Area A1 =SC00+UC164.SK008 - GF015 POWER CUT UC164 LINE
   "FDBACK_=SC00+UC16.EL001-Q32201/Q32202"(ON := "05_EM_STATE".A1_EMERGENCY_DELAY,   // FDBACK
                           FEEDBACK := "=SC00+UC16.EL001-Q32202 ( =SC00+UC164.SK008 - GF015 BELTS)",
                           QBAD_FIO := NOT "QBAD =SC00+UC16.EL001-Q32201/Q32202",
                           ACK_NEC := true,
                           ACK := "05_EM_STATE".A1_RESET,
                           FDB_TIME := T#300ms,
                           Q => "=SC00+UC16.EL001-Q32201 (=SC00+UC164.SK008 - GF015)");
END_REGION

REGION Network 93: Area A1 =SC00+UC164.GF016 - GF018 POWER CUT UC164 LINE
   "FDBACK_=SC00+UC16.EL001-Q32203/Q32204"(ON := "05_EM_STATE".A1_EMERGENCY_DELAY,   // FDBACK
                           FEEDBACK := "=SC00+UC16.EL001-Q32204 ( =SC00+UC164.GF016 - GF018 BELTS)",
                           QBAD_FIO := NOT "QBAD =SC00+UC16.EL001-Q32203/Q32204",
                           ACK_NEC := true,
                           ACK := "05_EM_STATE".A1_RESET,
                           FDB_TIME := T#300ms,
                           Q => "=SC00+UC16.EL001-Q32203 (=SC00+UC164.GF016 - GF018)");
END_REGION

REGION Network 94: Area A1 =SC00+UC165.GF001 - GF004 POWER CUT UC165 LINE
   "FDBACK_=SC00+UC16.EL001-Q32301/Q32302"(ON := "05_EM_STATE".A1_EMERGENCY_DELAY,   // FDBACK
                           FEEDBACK := "=SC00+UC16.EL001-Q32302 ( =SC00+UC165.GF001 - GF004 BELTS)",
                           QBAD_FIO := NOT "QBAD =SC00+UC16.EL001-Q32301/Q32302",
                           ACK_NEC := true,
                           ACK := "05_EM_STATE".A1_RESET,
                           FDB_TIME := T#300ms,
                           Q => "=SC00+UC16.EL001-Q32301 (=SC00+UC165.GF001 - GF004)");
END_REGION

REGION Network 95: Area A1 =SC00+UC166.GF001 - GF004 POWER CUT UC166 LINE
   "FDBACK_=SC00+UC16.EL001-Q32303/Q32304"(ON := "05_EM_STATE".A1_EMERGENCY_DELAY,   // FDBACK
                           FEEDBACK := "=SC00+UC16.EL001-Q32304 ( =SC00+UC166.GF001 - GF004 BELTS)",
                           QBAD_FIO := NOT "QBAD =SC00+UC16.EL001-Q32303/Q32304",
                           ACK_NEC := true,
                           ACK := "05_EM_STATE".A1_RESET,
                           FDB_TIME := T#300ms,
                           Q => "=SC00+UC16.EL001-Q32303 (=SC00+UC166.GF001 - GF004)");
END_REGION

REGION Network 96: Area A1 =SC00+UC167.RB001 - GF003 POWER CUT UC167 LINE
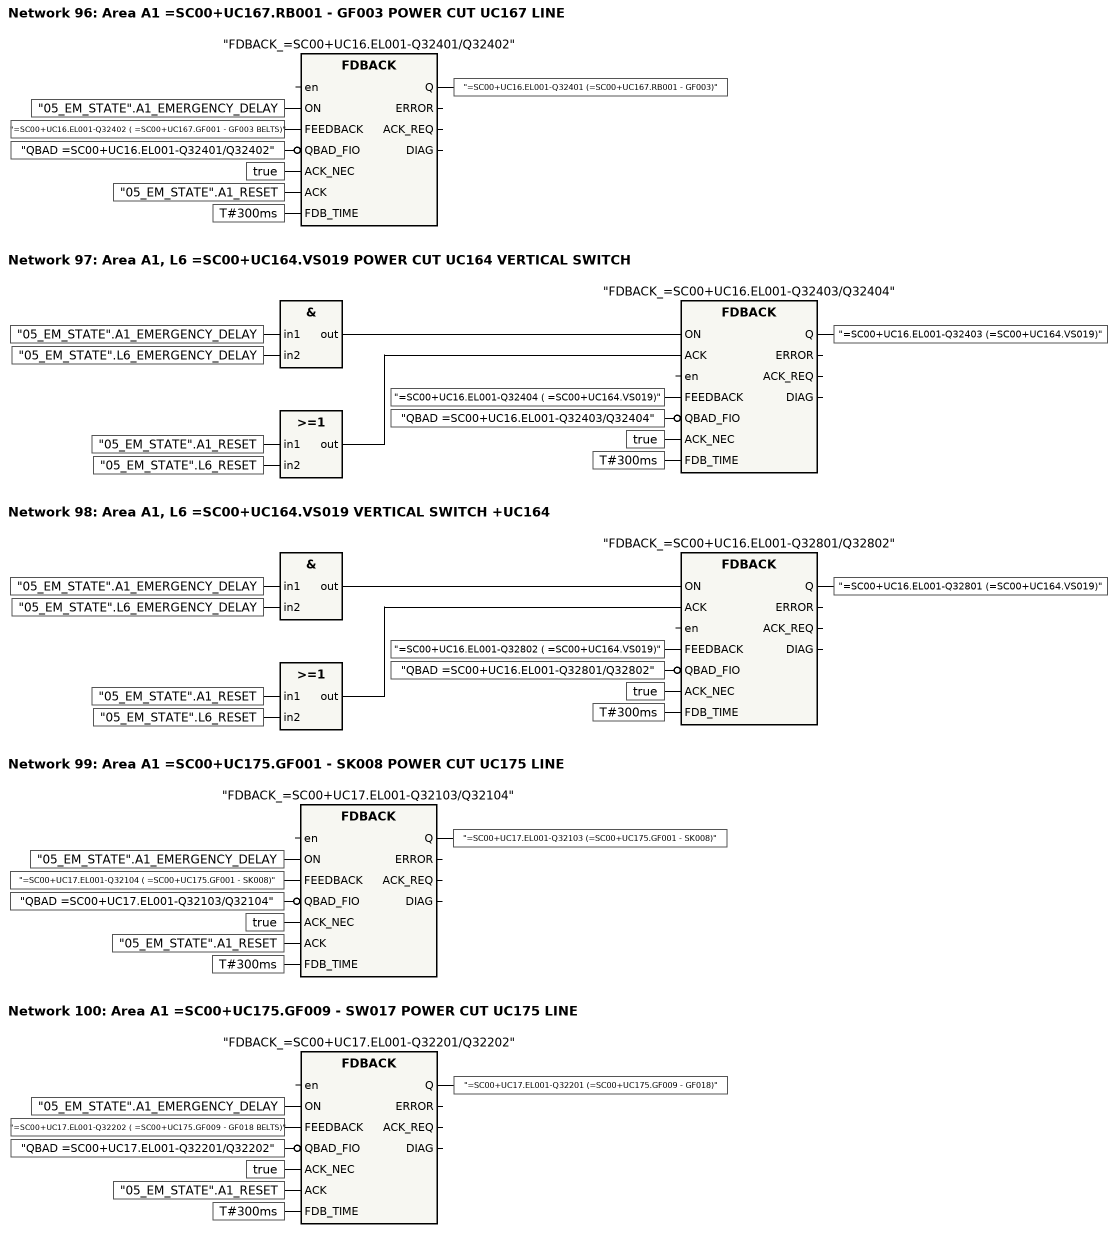
   "FDBACK_=SC00+UC16.EL001-Q32401/Q32402"(ON := "05_EM_STATE".A1_EMERGENCY_DELAY,   // FDBACK
                           FEEDBACK := "=SC00+UC16.EL001-Q32402 ( =SC00+UC167.GF001 - GF003 BELTS)",
                           QBAD_FIO := NOT "QBAD =SC00+UC16.EL001-Q32401/Q32402",
                           ACK_NEC := true,
                           ACK := "05_EM_STATE".A1_RESET,
                           FDB_TIME := T#300ms,
                           Q => "=SC00+UC16.EL001-Q32401 (=SC00+UC167.RB001 - GF003)");
END_REGION

REGION Network 97: Area A1, L6 =SC00+UC164.VS019 POWER CUT UC164 VERTICAL SWITCH
   "FDBACK_=SC00+UC16.EL001-Q32403/Q32404"(ON := "05_EM_STATE".A1_EMERGENCY_DELAY AND "05_EM_STATE".L6_EMERGENCY_DELAY,   // FDBACK
                           ACK := "05_EM_STATE".A1_RESET OR "05_EM_STATE".L6_RESET,
                           FEEDBACK := "=SC00+UC16.EL001-Q32404 ( =SC00+UC164.VS019)",
                           QBAD_FIO := NOT "QBAD =SC00+UC16.EL001-Q32403/Q32404",
                           ACK_NEC := true,
                           FDB_TIME := T#300ms,
                           Q => "=SC00+UC16.EL001-Q32403 (=SC00+UC164.VS019)");
END_REGION

REGION Network 98: Area A1, L6 =SC00+UC164.VS019 VERTICAL SWITCH +UC164
   "FDBACK_=SC00+UC16.EL001-Q32801/Q32802"(ON := "05_EM_STATE".A1_EMERGENCY_DELAY AND "05_EM_STATE".L6_EMERGENCY_DELAY,   // FDBACK
                           ACK := "05_EM_STATE".A1_RESET OR "05_EM_STATE".L6_RESET,
                           FEEDBACK := "=SC00+UC16.EL001-Q32802 ( =SC00+UC164.VS019)",
                           QBAD_FIO := NOT "QBAD =SC00+UC16.EL001-Q32801/Q32802",
                           ACK_NEC := true,
                           FDB_TIME := T#300ms,
                           Q => "=SC00+UC16.EL001-Q32801 (=SC00+UC164.VS019)");
END_REGION

REGION Network 99: Area A1 =SC00+UC175.GF001 - SK008 POWER CUT UC175 LINE
   "FDBACK_=SC00+UC17.EL001-Q32103/Q32104"(ON := "05_EM_STATE".A1_EMERGENCY_DELAY,   // FDBACK
                           FEEDBACK := "=SC00+UC17.EL001-Q32104 ( =SC00+UC175.GF001 - SK008)",
                           QBAD_FIO := NOT "QBAD =SC00+UC17.EL001-Q32103/Q32104",
                           ACK_NEC := true,
                           ACK := "05_EM_STATE".A1_RESET,
                           FDB_TIME := T#300ms,
                           Q => "=SC00+UC17.EL001-Q32103 (=SC00+UC175.GF001 - SK008)");
END_REGION

REGION Network 100: Area A1 =SC00+UC175.GF009 - SW017 POWER CUT UC175 LINE
   "FDBACK_=SC00+UC17.EL001-Q32201/Q32202"(ON := "05_EM_STATE".A1_EMERGENCY_DELAY,   // FDBACK
                           FEEDBACK := "=SC00+UC17.EL001-Q32202 ( =SC00+UC175.GF009 - GF018 BELTS)",
                           QBAD_FIO := NOT "QBAD =SC00+UC17.EL001-Q32201/Q32202",
                           ACK_NEC := true,
                           ACK := "05_EM_STATE".A1_RESET,
                           FDB_TIME := T#300ms,
                           Q => "=SC00+UC17.EL001-Q32201 (=SC00+UC175.GF009 - GF018)");
END_REGION

REGION Network 101: Area A1 =SC00+UC176.GF001 - GF004 POWER CUT UC176 LINE
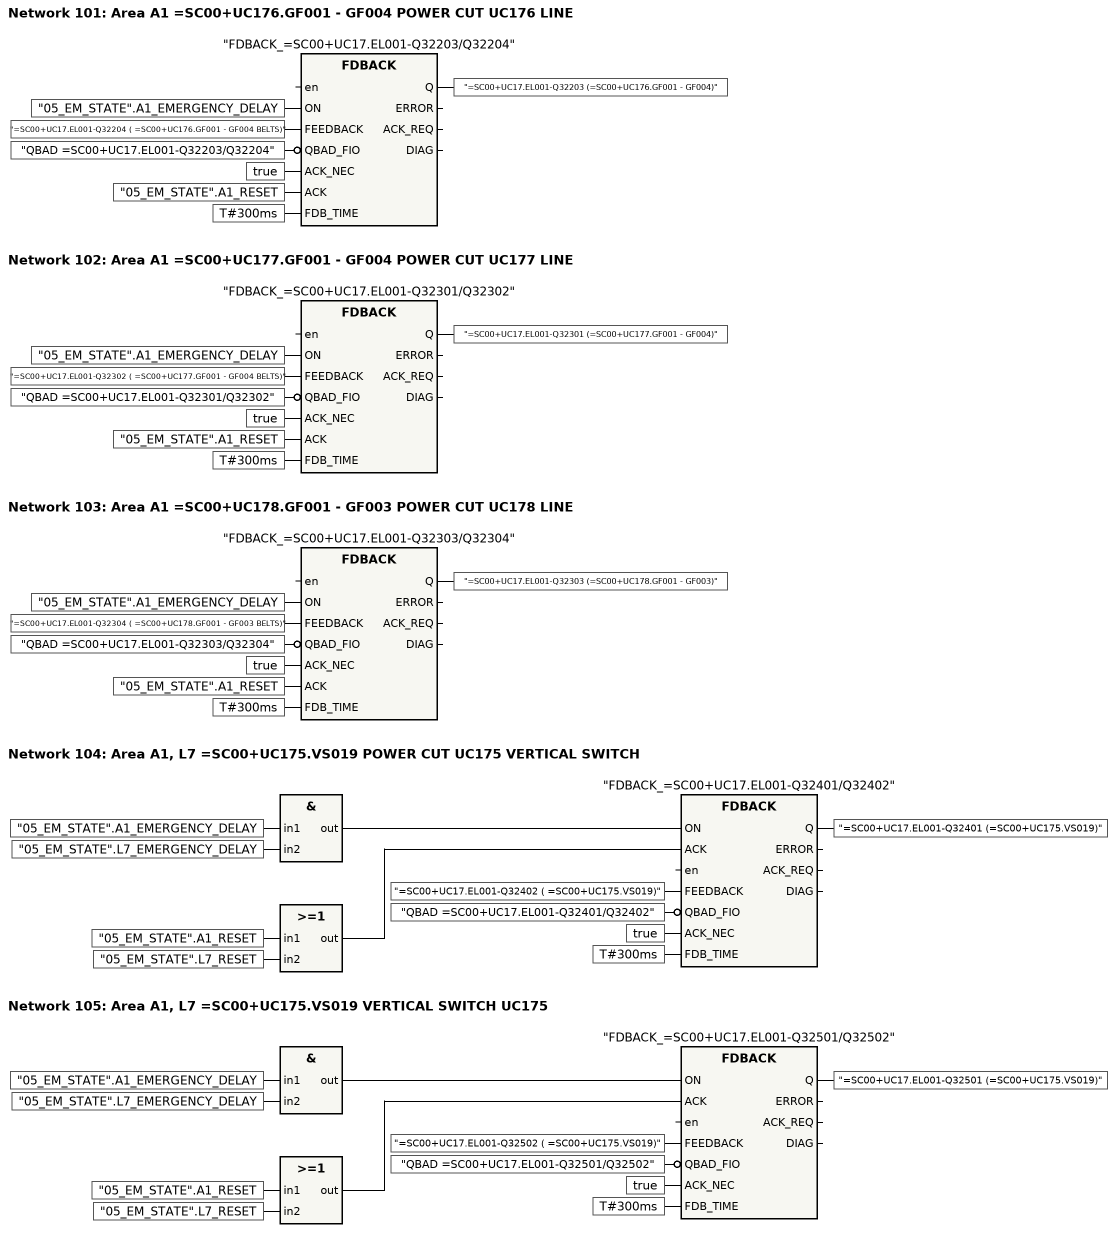
   "FDBACK_=SC00+UC17.EL001-Q32203/Q32204"(ON := "05_EM_STATE".A1_EMERGENCY_DELAY,   // FDBACK
                           FEEDBACK := "=SC00+UC17.EL001-Q32204 ( =SC00+UC176.GF001 - GF004 BELTS)",
                           QBAD_FIO := NOT "QBAD =SC00+UC17.EL001-Q32203/Q32204",
                           ACK_NEC := true,
                           ACK := "05_EM_STATE".A1_RESET,
                           FDB_TIME := T#300ms,
                           Q => "=SC00+UC17.EL001-Q32203 (=SC00+UC176.GF001 - GF004)");
END_REGION

REGION Network 102: Area A1 =SC00+UC177.GF001 - GF004 POWER CUT UC177 LINE
   "FDBACK_=SC00+UC17.EL001-Q32301/Q32302"(ON := "05_EM_STATE".A1_EMERGENCY_DELAY,   // FDBACK
                           FEEDBACK := "=SC00+UC17.EL001-Q32302 ( =SC00+UC177.GF001 - GF004 BELTS)",
                           QBAD_FIO := NOT "QBAD =SC00+UC17.EL001-Q32301/Q32302",
                           ACK_NEC := true,
                           ACK := "05_EM_STATE".A1_RESET,
                           FDB_TIME := T#300ms,
                           Q => "=SC00+UC17.EL001-Q32301 (=SC00+UC177.GF001 - GF004)");
END_REGION

REGION Network 103: Area A1 =SC00+UC178.GF001 - GF003 POWER CUT UC178 LINE
   "FDBACK_=SC00+UC17.EL001-Q32303/Q32304"(ON := "05_EM_STATE".A1_EMERGENCY_DELAY,   // FDBACK
                           FEEDBACK := "=SC00+UC17.EL001-Q32304 ( =SC00+UC178.GF001 - GF003 BELTS)",
                           QBAD_FIO := NOT "QBAD =SC00+UC17.EL001-Q32303/Q32304",
                           ACK_NEC := true,
                           ACK := "05_EM_STATE".A1_RESET,
                           FDB_TIME := T#300ms,
                           Q => "=SC00+UC17.EL001-Q32303 (=SC00+UC178.GF001 - GF003)");
END_REGION

REGION Network 104: Area A1, L7 =SC00+UC175.VS019 POWER CUT UC175 VERTICAL SWITCH
   "FDBACK_=SC00+UC17.EL001-Q32401/Q32402"(ON := "05_EM_STATE".A1_EMERGENCY_DELAY AND "05_EM_STATE".L7_EMERGENCY_DELAY,   // FDBACK
                           ACK := "05_EM_STATE".A1_RESET OR "05_EM_STATE".L7_RESET,
                           FEEDBACK := "=SC00+UC17.EL001-Q32402 ( =SC00+UC175.VS019)",
                           QBAD_FIO := NOT "QBAD =SC00+UC17.EL001-Q32401/Q32402",
                           ACK_NEC := true,
                           FDB_TIME := T#300ms,
                           Q => "=SC00+UC17.EL001-Q32401 (=SC00+UC175.VS019)");
END_REGION

REGION Network 105: Area A1, L7 =SC00+UC175.VS019 VERTICAL SWITCH UC175
   "FDBACK_=SC00+UC17.EL001-Q32501/Q32502"(ON := "05_EM_STATE".A1_EMERGENCY_DELAY AND "05_EM_STATE".L7_EMERGENCY_DELAY,   // FDBACK
                           ACK := "05_EM_STATE".A1_RESET OR "05_EM_STATE".L7_RESET,
                           FEEDBACK := "=SC00+UC17.EL001-Q32502 ( =SC00+UC175.VS019)",
                           QBAD_FIO := NOT "QBAD =SC00+UC17.EL001-Q32501/Q32502",
                           ACK_NEC := true,
                           FDB_TIME := T#300ms,
                           Q => "=SC00+UC17.EL001-Q32501 (=SC00+UC175.VS019)");
END_REGION

REGION Network 106: Area A2 =SF00+UF317.GF001 - GF012 POWER CUT UF317 LINE
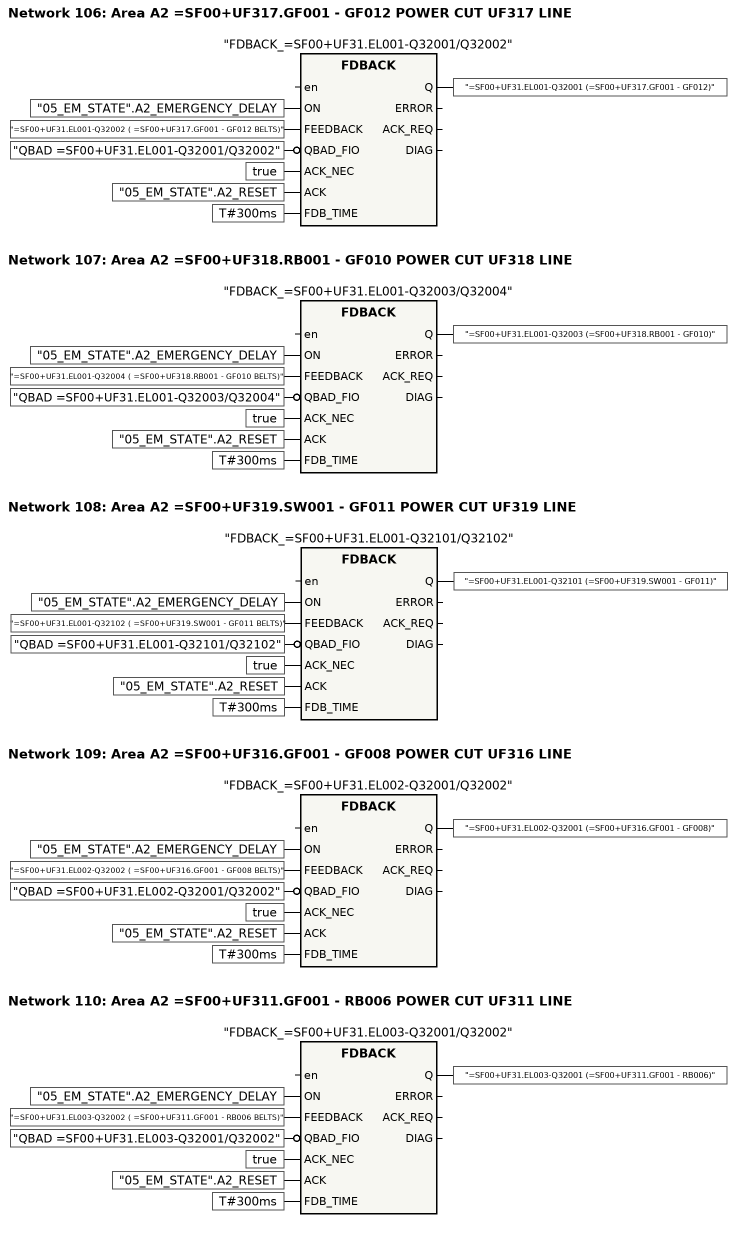
   "FDBACK_=SF00+UF31.EL001-Q32001/Q32002"(ON := "05_EM_STATE".A2_EMERGENCY_DELAY,   // FDBACK
                           FEEDBACK := "=SF00+UF31.EL001-Q32002 ( =SF00+UF317.GF001 - GF012 BELTS)",
                           QBAD_FIO := NOT "QBAD =SF00+UF31.EL001-Q32001/Q32002",
                           ACK_NEC := true,
                           ACK := "05_EM_STATE".A2_RESET,
                           FDB_TIME := T#300ms,
                           Q => "=SF00+UF31.EL001-Q32001 (=SF00+UF317.GF001 - GF012)");
END_REGION

REGION Network 107: Area A2 =SF00+UF318.RB001 - GF010 POWER CUT UF318 LINE
   "FDBACK_=SF00+UF31.EL001-Q32003/Q32004"(ON := "05_EM_STATE".A2_EMERGENCY_DELAY,   // FDBACK
                           FEEDBACK := "=SF00+UF31.EL001-Q32004 ( =SF00+UF318.RB001 - GF010 BELTS)",
                           QBAD_FIO := NOT "QBAD =SF00+UF31.EL001-Q32003/Q32004",
                           ACK_NEC := true,
                           ACK := "05_EM_STATE".A2_RESET,
                           FDB_TIME := T#300ms,
                           Q => "=SF00+UF31.EL001-Q32003 (=SF00+UF318.RB001 - GF010)");
END_REGION

REGION Network 108: Area A2 =SF00+UF319.SW001 - GF011 POWER CUT UF319 LINE
   "FDBACK_=SF00+UF31.EL001-Q32101/Q32102"(ON := "05_EM_STATE".A2_EMERGENCY_DELAY,   // FDBACK
                           FEEDBACK := "=SF00+UF31.EL001-Q32102 ( =SF00+UF319.SW001 - GF011 BELTS)",
                           QBAD_FIO := NOT "QBAD =SF00+UF31.EL001-Q32101/Q32102",
                           ACK_NEC := true,
                           ACK := "05_EM_STATE".A2_RESET,
                           FDB_TIME := T#300ms,
                           Q => "=SF00+UF31.EL001-Q32101 (=SF00+UF319.SW001 - GF011)");
END_REGION

REGION Network 109: Area A2 =SF00+UF316.GF001 - GF008 POWER CUT UF316 LINE
   "FDBACK_=SF00+UF31.EL002-Q32001/Q32002"(ON := "05_EM_STATE".A2_EMERGENCY_DELAY,   // FDBACK
                           FEEDBACK := "=SF00+UF31.EL002-Q32002 ( =SF00+UF316.GF001 - GF008 BELTS)",
                           QBAD_FIO := NOT "QBAD =SF00+UF31.EL002-Q32001/Q32002",
                           ACK_NEC := true,
                           ACK := "05_EM_STATE".A2_RESET,
                           FDB_TIME := T#300ms,
                           Q => "=SF00+UF31.EL002-Q32001 (=SF00+UF316.GF001 - GF008)");
END_REGION

REGION Network 110: Area A2 =SF00+UF311.GF001 - RB006 POWER CUT UF311 LINE
   "FDBACK_=SF00+UF31.EL003-Q32001/Q32002"(ON := "05_EM_STATE".A2_EMERGENCY_DELAY,   // FDBACK
                           FEEDBACK := "=SF00+UF31.EL003-Q32002 ( =SF00+UF311.GF001 - RB006 BELTS)",
                           QBAD_FIO := NOT "QBAD =SF00+UF31.EL003-Q32001/Q32002",
                           ACK_NEC := true,
                           ACK := "05_EM_STATE".A2_RESET,
                           FDB_TIME := T#300ms,
                           Q => "=SF00+UF31.EL003-Q32001 (=SF00+UF311.GF001 - RB006)");
END_REGION

REGION Network 111: Area A2 =SF00+UF312.GF001 - RB006 POWER CUT UF312 LINE
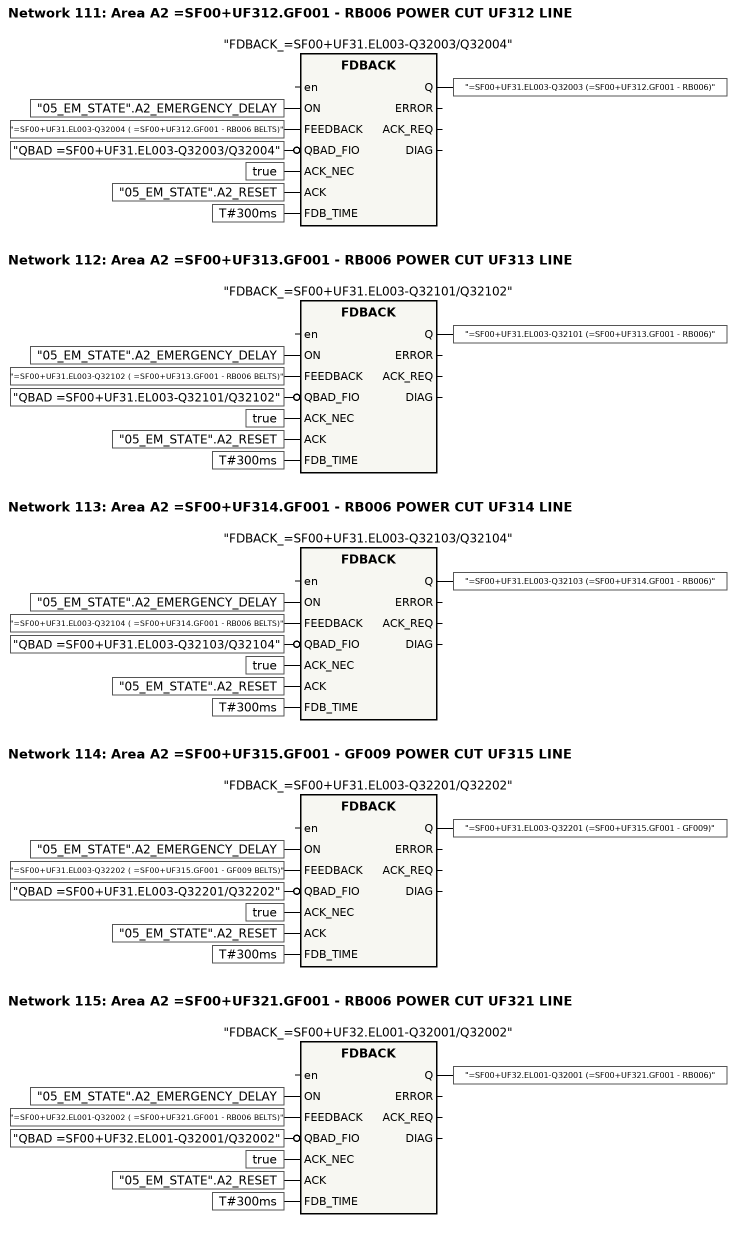
   "FDBACK_=SF00+UF31.EL003-Q32003/Q32004"(ON := "05_EM_STATE".A2_EMERGENCY_DELAY,   // FDBACK
                           FEEDBACK := "=SF00+UF31.EL003-Q32004 ( =SF00+UF312.GF001 - RB006 BELTS)",
                           QBAD_FIO := NOT "QBAD =SF00+UF31.EL003-Q32003/Q32004",
                           ACK_NEC := true,
                           ACK := "05_EM_STATE".A2_RESET,
                           FDB_TIME := T#300ms,
                           Q => "=SF00+UF31.EL003-Q32003 (=SF00+UF312.GF001 - RB006)");
END_REGION

REGION Network 112: Area A2 =SF00+UF313.GF001 - RB006 POWER CUT UF313 LINE
   "FDBACK_=SF00+UF31.EL003-Q32101/Q32102"(ON := "05_EM_STATE".A2_EMERGENCY_DELAY,   // FDBACK
                           FEEDBACK := "=SF00+UF31.EL003-Q32102 ( =SF00+UF313.GF001 - RB006 BELTS)",
                           QBAD_FIO := NOT "QBAD =SF00+UF31.EL003-Q32101/Q32102",
                           ACK_NEC := true,
                           ACK := "05_EM_STATE".A2_RESET,
                           FDB_TIME := T#300ms,
                           Q => "=SF00+UF31.EL003-Q32101 (=SF00+UF313.GF001 - RB006)");
END_REGION

REGION Network 113: Area A2 =SF00+UF314.GF001 - RB006 POWER CUT UF314 LINE
   "FDBACK_=SF00+UF31.EL003-Q32103/Q32104"(ON := "05_EM_STATE".A2_EMERGENCY_DELAY,   // FDBACK
                           FEEDBACK := "=SF00+UF31.EL003-Q32104 ( =SF00+UF314.GF001 - RB006 BELTS)",
                           QBAD_FIO := NOT "QBAD =SF00+UF31.EL003-Q32103/Q32104",
                           ACK_NEC := true,
                           ACK := "05_EM_STATE".A2_RESET,
                           FDB_TIME := T#300ms,
                           Q => "=SF00+UF31.EL003-Q32103 (=SF00+UF314.GF001 - RB006)");
END_REGION

REGION Network 114: Area A2 =SF00+UF315.GF001 - GF009 POWER CUT UF315 LINE
   "FDBACK_=SF00+UF31.EL003-Q32201/Q32202"(ON := "05_EM_STATE".A2_EMERGENCY_DELAY,   // FDBACK
                           FEEDBACK := "=SF00+UF31.EL003-Q32202 ( =SF00+UF315.GF001 - GF009 BELTS)",
                           QBAD_FIO := NOT "QBAD =SF00+UF31.EL003-Q32201/Q32202",
                           ACK_NEC := true,
                           ACK := "05_EM_STATE".A2_RESET,
                           FDB_TIME := T#300ms,
                           Q => "=SF00+UF31.EL003-Q32201 (=SF00+UF315.GF001 - GF009)");
END_REGION

REGION Network 115: Area A2 =SF00+UF321.GF001 - RB006 POWER CUT UF321 LINE
   "FDBACK_=SF00+UF32.EL001-Q32001/Q32002"(ON := "05_EM_STATE".A2_EMERGENCY_DELAY,   // FDBACK
                           FEEDBACK := "=SF00+UF32.EL001-Q32002 ( =SF00+UF321.GF001 - RB006 BELTS)",
                           QBAD_FIO := NOT "QBAD =SF00+UF32.EL001-Q32001/Q32002",
                           ACK_NEC := true,
                           ACK := "05_EM_STATE".A2_RESET,
                           FDB_TIME := T#300ms,
                           Q => "=SF00+UF32.EL001-Q32001 (=SF00+UF321.GF001 - RB006)");
END_REGION

REGION Network 116: Area A2 =SF00+UF322.GF001 - RB006 POWER CUT UF322 LINE
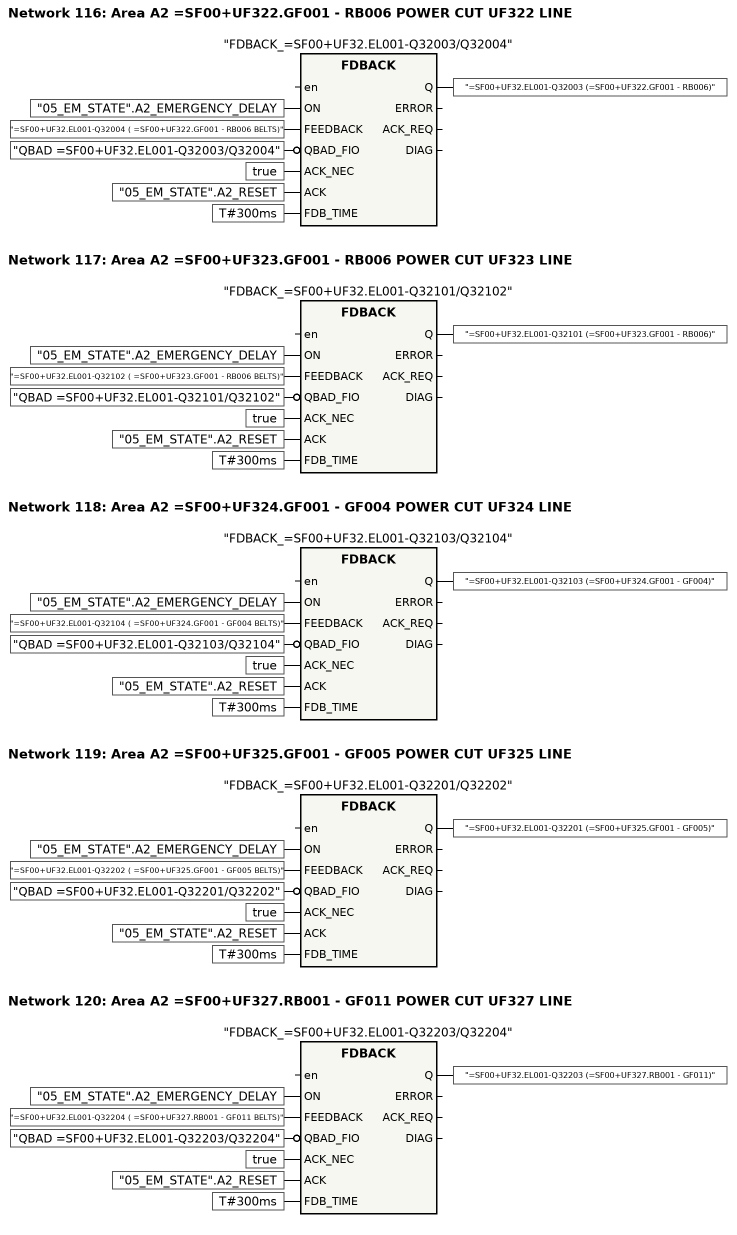
   "FDBACK_=SF00+UF32.EL001-Q32003/Q32004"(ON := "05_EM_STATE".A2_EMERGENCY_DELAY,   // FDBACK
                           FEEDBACK := "=SF00+UF32.EL001-Q32004 ( =SF00+UF322.GF001 - RB006 BELTS)",
                           QBAD_FIO := NOT "QBAD =SF00+UF32.EL001-Q32003/Q32004",
                           ACK_NEC := true,
                           ACK := "05_EM_STATE".A2_RESET,
                           FDB_TIME := T#300ms,
                           Q => "=SF00+UF32.EL001-Q32003 (=SF00+UF322.GF001 - RB006)");
END_REGION

REGION Network 117: Area A2 =SF00+UF323.GF001 - RB006 POWER CUT UF323 LINE
   "FDBACK_=SF00+UF32.EL001-Q32101/Q32102"(ON := "05_EM_STATE".A2_EMERGENCY_DELAY,   // FDBACK
                           FEEDBACK := "=SF00+UF32.EL001-Q32102 ( =SF00+UF323.GF001 - RB006 BELTS)",
                           QBAD_FIO := NOT "QBAD =SF00+UF32.EL001-Q32101/Q32102",
                           ACK_NEC := true,
                           ACK := "05_EM_STATE".A2_RESET,
                           FDB_TIME := T#300ms,
                           Q => "=SF00+UF32.EL001-Q32101 (=SF00+UF323.GF001 - RB006)");
END_REGION

REGION Network 118: Area A2 =SF00+UF324.GF001 - GF004 POWER CUT UF324 LINE
   "FDBACK_=SF00+UF32.EL001-Q32103/Q32104"(ON := "05_EM_STATE".A2_EMERGENCY_DELAY,   // FDBACK
                           FEEDBACK := "=SF00+UF32.EL001-Q32104 ( =SF00+UF324.GF001 - GF004 BELTS)",
                           QBAD_FIO := NOT "QBAD =SF00+UF32.EL001-Q32103/Q32104",
                           ACK_NEC := true,
                           ACK := "05_EM_STATE".A2_RESET,
                           FDB_TIME := T#300ms,
                           Q => "=SF00+UF32.EL001-Q32103 (=SF00+UF324.GF001 - GF004)");
END_REGION

REGION Network 119: Area A2 =SF00+UF325.GF001 - GF005 POWER CUT UF325 LINE
   "FDBACK_=SF00+UF32.EL001-Q32201/Q32202"(ON := "05_EM_STATE".A2_EMERGENCY_DELAY,   // FDBACK
                           FEEDBACK := "=SF00+UF32.EL001-Q32202 ( =SF00+UF325.GF001 - GF005 BELTS)",
                           QBAD_FIO := NOT "QBAD =SF00+UF32.EL001-Q32201/Q32202",
                           ACK_NEC := true,
                           ACK := "05_EM_STATE".A2_RESET,
                           FDB_TIME := T#300ms,
                           Q => "=SF00+UF32.EL001-Q32201 (=SF00+UF325.GF001 - GF005)");
END_REGION

REGION Network 120: Area A2 =SF00+UF327.RB001 - GF011 POWER CUT UF327 LINE
   "FDBACK_=SF00+UF32.EL001-Q32203/Q32204"(ON := "05_EM_STATE".A2_EMERGENCY_DELAY,   // FDBACK
                           FEEDBACK := "=SF00+UF32.EL001-Q32204 ( =SF00+UF327.RB001 - GF011 BELTS)",
                           QBAD_FIO := NOT "QBAD =SF00+UF32.EL001-Q32203/Q32204",
                           ACK_NEC := true,
                           ACK := "05_EM_STATE".A2_RESET,
                           FDB_TIME := T#300ms,
                           Q => "=SF00+UF32.EL001-Q32203 (=SF00+UF327.RB001 - GF011)");
END_REGION

REGION Network 121: Area A2 =SF00+UF327.SW001 - GF011 POWER CUT UF327 LINE
